# B&R Automation Studio project GAT (part 6)

#### RecipeMgt.typ - Local data types
```iecst
TYPE
	RecipeCommands_type : 	STRUCT
		StoreMachineSettings : BOOL;
		FactoryResetMachineSettings : BOOL;
		SaveCurrentRecipe : BOOL;
		ImportFromUSB : BOOL;
		ExportToUSB : BOOL;
		SaveSelectedRecipe : BOOL;
		LoadRecipe : BOOL;
		CreateRecipe : BOOL;
	END_STRUCT;
	RecipeParameters_type : 	STRUCT
		Category : STRING[30];
		LastLoadedConfigRecipe : STRING[255];
		LastLoadedProductRecipe : STRING[255];
		ActiveRecipe : STRING[255];
		DeviceDataProvider : ARRAY[0..MAX_IDX_FILE_DEV]OF STRING[100];
		DeviceName : STRING[50];
		FileName : STRING[255];
		LastSelectedIndex : UINT;
		LastStatus : MpRecipeUIStatusEnum;
		TableConfig : STRING[120];
		CopyStep : RecipeCopyStep_enum;
		CategoryDropdown : STRING[50];
		EditDialogOpened : BOOL;
		CreateDialogOpened : BOOL;
	END_STRUCT;
	RecipeStatus_type : 	STRUCT
		HMIcommand : RecipeHmiStep_enum;
	END_STRUCT;
	RecipeHmiInterface_type : 	STRUCT
		Commands : RecipeCommands_type;
		Parameters : RecipeParameters_type;
		Status : RecipeStatus_type;
	END_STRUCT;
	RecipeCopyStep_enum :
		(
		REC_COPY_WAIT := 0,
		REC_COPY_TO_USB,
		REC_COPY_FROM_USB,
		REC_COPY_BUSY
		);
	MachineSettings_type : 	STRUCT
		AddMachineSettingsHere1 : USINT;
		AddMachineSettingsHere2 : DINT;
		AddMachineSettingsHere3 : BOOL;
		AddMachineSettingsHere4 : REAL;
		AddMachineSettingsHere5 : UINT;
	END_STRUCT;
	Parameters_type : 	STRUCT
		AddParametersHere1 : BOOL;
		AddParametersHere2 : STRING[80];
		AddParametersHere3 : REAL;
		AddParametersHere4 : REAL;
		AddParametersHere5 : REAL;
	END_STRUCT;
	RecipeHmiStep_enum :
		(
		REC_HMI_WAIT,
		REC_HMI_LOAD,
		REC_HMI_SAVE,
		REC_HMI_CREATE
		);
END_TYPE
```

#### RecipeMgt.var - Local variables
```iecst
(********************************************************************
 * COPYRIGHT -- Bernecker + Rainer
 ********************************************************************
 * Program: FolderHandling
 * File: FolderHandling.var
 * Author: Bernecker + Rainer
 * Created: December , 2020
 ********************************************************************
 * Local variables of program AlarmManagement
 ********************************************************************)
(*Function Block Declaration*)
VAR
	MpRecipe_0 : MpRecipeXml; (*Recipe Management Function Block*)
	MpRecipeUI_0 : MpRecipeUI; (*Recipe to UI*)
	DirCreate_New : DirCreate;
END_VAR
(*Recipe Management Variables*)
VAR
	Index : USINT; (*Index to loop through file devices*)
	MpRecipeUISetup : MpRecipeUISetupType; (*MpRecipeUI connection datapoints*) (*ParameterFileStep : INT;*)
	MpRecipeUIConnect : MpRecipeUIConnectType; (*MpRecipeUI connection datapoints*) (*ParameterFileStep : INT;*)
	HmiRecipe : RecipeHmiInterfaceType;
	Header : MpRecipeXmlHeaderType;
	DTGetTime_0 : DTGetTime;
END_VAR
(*File Management Variables*)
VAR
	MpFileManagerUIConnect : MpFileManagerUIConnectType;
	MpFileManagerUI_0 : MpFileManagerUI;
END_VAR
(*Defines*)
VAR CONSTANT
	MAX_IDX_FILE_DEV : USINT := MAX_IDX_USB_DEV_LIST + 1;
	MACHINE_FILENAME : STRING[12] := 'Machine.mcfg';
	LOCAL_FOLDER : STRING[10] := 'Recipe';
END_VAR
VAR
	MpRecipeRegPar_PreviewPar : MpRecipeRegPar;
	MpRecipeRegPar_PreviewCfg : MpRecipeRegPar;
	Parameters : ParametersType;
	ParametersEdit : {REDUND_UNREPLICABLE} ParametersType;
	ParametersPreview : ParametersType;
	MachineSettings : MachineSettingsType;
	MachineSettingsEdit : MachineSettingsType;
	MachineSettingsPreview : MachineSettingsType;
	PreviousRecipe : STRING[80];
END_VAR
```

#### HMIActions.st
```iecst
ACTION FormatDeviceDataProvider:

	// Select CF device if USB device is not available
	FOR Index := 0 TO MAX_IDX_USB_DEV_LIST DO
		IF gUSBAvailable[Index] THEN
			HmiRecipe.Parameters.DeviceDataProvider[Index + 1] := '{"value":"USB';
			brsitoa(Index + 1, ADR(HmiRecipe.Parameters.DeviceDataProvider[Index + 1]) + brsstrlen(ADR(HmiRecipe.Parameters.DeviceDataProvider[Index + 1])));
			brsstrcat(ADR(HmiRecipe.Parameters.DeviceDataProvider[Index + 1]), ADR('","text":"USB'));
			brsitoa(Index + 1, ADR(HmiRecipe.Parameters.DeviceDataProvider[Index + 1]) + brsstrlen(ADR(HmiRecipe.Parameters.DeviceDataProvider[Index + 1])));
			brsstrcat(ADR(HmiRecipe.Parameters.DeviceDataProvider[Index + 1]), ADR('"}'));
			brsstrcpy(ADR(MpFileManagerUIConnect.DeviceList.DeviceNames[Index + 1]), ADR('USB'));
			brsitoa(Index + 1, ADR(MpFileManagerUIConnect.DeviceList.DeviceNames[Index + 1]) + brsstrlen(ADR(MpFileManagerUIConnect.DeviceList.DeviceNames[Index + 1])));
		ELSE
			brsmemset(ADR(HmiRecipe.Parameters.DeviceDataProvider[Index + 1]), 0, SIZEOF(HmiRecipe.Parameters.DeviceDataProvider[Index + 1]));
			brsmemset(ADR(MpFileManagerUIConnect.DeviceList.DeviceNames[Index + 1]), 0, SIZEOF(MpFileManagerUIConnect.DeviceList.DeviceNames[Index + 1]));
		END_IF
	END_FOR

	// Configure visible recipe list
	HmiRecipe.Parameters.TableConfig := '{ "specRows": [{"from":';
	brsitoa(MpRecipeUIConnect.Recipe.List.MaxSelection + 1, ADR(HmiRecipe.Parameters.TableConfig) + brsstrlen(ADR(HmiRecipe.Parameters.TableConfig)));
	brsstrcat(ADR(HmiRecipe.Parameters.TableConfig),  ADR(',"to":19, "visible":false}]}'));

END_ACTION

ACTION LoadPreview:

	// Load preview when a recipe is selected
	IF (MpRecipeUIConnect.Recipe.List.SelectedIndex <> HmiRecipe.Parameters.LastSelectedIndex) THEN
		// Check selected recipe name is not empty
		IF (brsstrlen(ADR(MpRecipeUIConnect.Recipe.List.Names[MpRecipeUIConnect.Recipe.List.SelectedIndex])) > 0) THEN
			MpRecipe_0.FileName := ADR(MpRecipeUIConnect.Recipe.List.Names[MpRecipeUIConnect.Recipe.List.SelectedIndex]);
			MpRecipe_0.Category := ADR(HmiRecipe.Parameters.CategoryDropdown);
			MpRecipe_0.Load := TRUE;
			HmiRecipe.Parameters.LastSelectedIndex := MpRecipeUIConnect.Recipe.List.SelectedIndex;
		END_IF
	END_IF

	// Reset load command on MpRecipe_Pre FUB
	IF ((MpRecipe_0.CommandDone = TRUE) OR (MpRecipe_0.Error = TRUE)) THEN
		MpRecipe_0.Load := FALSE;
	END_IF

END_ACTION

ACTION RecipeHMIcommands:

    CASE HmiRecipe.Status.HMIcommand OF
        REC_HMI_WAIT:
            IF HmiRecipe.Commands.CreateRecipe THEN
				HmiRecipe.Status.HMIcommand := REC_HMI_CREATE;
				HmiRecipe.Commands.CreateRecipe := FALSE;
			ELSIF HmiRecipe.Commands.SaveSelectedRecipe THEN
				HmiRecipe.Status.HMIcommand := REC_HMI_SAVE;
				HmiRecipe.Commands.SaveSelectedRecipe := FALSE;
			ELSIF HmiRecipe.Commands.LoadRecipe THEN
				HmiRecipe.Status.HMIcommand := REC_HMI_LOAD;
				HmiRecipe.Commands.LoadRecipe := FALSE;
			END_IF

		REC_HMI_CREATE:
			IF (brsstrcmp(ADR(HmiRecipe.Parameters.CategoryDropdown),ADR('Product')) = 0) THEN
				ParametersPreview := ParametersEdit;
			ELSIF (brsstrcmp(ADR(HmiRecipe.Parameters.CategoryDropdown),ADR('Machine')) = 0) THEN
				MachSettingsPreview := MachSettingsEdit;
			END_IF
			MpRecipeUIConnect.New.Create := TRUE;
			HmiRecipe.Status.HMIcommand := REC_HMI_WAIT;

		REC_HMI_LOAD:
			IF (brsstrcmp(ADR(HmiRecipe.Parameters.CategoryDropdown),ADR('Product')) = 0) THEN
				Parameters := ParametersPreview;
				HmiRecipe.Parameters.LastLoadedProductRecipe := HmiRecipe.Parameters.ActiveRecipe;
			ELSIF (brsstrcmp(ADR(HmiRecipe.Parameters.CategoryDropdown),ADR('Machine')) = 0) THEN
				MachSettings := MachSettingsPreview;
				HmiRecipe.Parameters.LastLoadedConfigRecipe := HmiRecipe.Parameters.ActiveRecipe;
			END_IF
			HmiRecipe.Status.HMIcommand := REC_HMI_WAIT;

		REC_HMI_SAVE:
			IF (brsstrcmp(ADR(HmiRecipe.Parameters.CategoryDropdown),ADR('Product')) = 0) THEN
				ParametersPreview := ParametersEdit;
	        ELSIF (brsstrcmp(ADR(HmiRecipe.Parameters.CategoryDropdown),ADR('Machine')) = 0) THEN
                MachSettingsPreview := MachSettingsEdit;
            END_IF

            IF (brsstrlen(ADR(HmiRecipe.Parameters.ActiveRecipe)) > 0) THEN
                MpRecipe_0.FileName := ADR(HmiRecipe.Parameters.ActiveRecipe);
				MpRecipe_0.Save := TRUE;
			END_IF
			HmiRecipe.Status.HMIcommand := REC_HMI_WAIT;

	END_CASE

	IF NOT MpRecipe_0.CommandBusy AND brsstrcmp(ADR(PreviousRecipe),ADR(HmiRecipe.Parameters.FileName)) <> 0 THEN
		HmiRecipe.Parameters.FileName := PreviousRecipe;
	END_IF

	IF HmiRecipe.Parameters.EditDialogOpened OR HmiRecipe.Parameters.CreateDialogOpened THEN
		IF (brsstrcmp(ADR(HmiRecipe.Parameters.CategoryDropdown),ADR('Product')) = 0) THEN
			ParametersEdit := ParametersPreview;
			MpRecipeUIConnect.New.FileName := 'newParameters.par';
		ELSIF (brsstrcmp(ADR(HmiRecipe.Parameters.CategoryDropdown),ADR('Machine')) = 0) THEN
			MachSettingsEdit := MachSettingsPreview;
			MpRecipeUIConnect.New.FileName := 'newMachConfig.mcfg';
		END_IF
		HmiRecipe.Parameters.EditDialogOpened := FALSE;
		HmiRecipe.Parameters.CreateDialogOpened := FALSE;
	END_IF

END_ACTION
```

#### FileOperations.st
```iecst
ACTION FileCopyOperation:

	// Export/Import recipes to/from USB
    CASE HmiRecipe.Parameters.CopyStep OF
		REC_COPY_WAIT:
			//Wait for export/import command
            IF (HmiRecipe.Commands.ExportToUSB = TRUE) THEN
                // Check if USB device is available
                IF (brsstrlen(ADR(MpFileManagerUIConnect.DeviceList.DeviceNames[1])) > 0) THEN
					// USB is available proceed with export: select all files on the CF and trigger copy command
                    IF (MpFileManagerUIConnect.DeviceList.SelectedIndex <> 0) THEN
                        MpFileManagerUIConnect.DeviceList.SelectedIndex := 0;
                        MpFileManagerUIConnect.File.MultiSelect := FALSE;
                    ELSIF (MpFileManagerUIConnect.Status = mpFILE_UI_STATUS_IDLE) THEN

                        IF NOT MpFileManagerUIConnect.File.MultiSelect THEN
                            MpFileManagerUIConnect.File.MultiSelect := TRUE;
                            FOR Index := 0 TO 49 DO
                                MpFileManagerUIConnect.File.List.Items[Index].IsSelected := TRUE;
                            END_FOR
                        ELSIF (brsstrlen(ADR(MpFileManagerUIConnect.File.List.Items[Index].Name)) = 0) THEN
                            // No files to copy, cancel operation
                            HmiRecipe.Commands.ExportToUSB := FALSE;
                        ELSE
                            MpFileManagerUIConnect.File.Copy := TRUE;
							HmiRecipe.Parameters.CopyStep := REC_COPY_TO_USB;
                            HmiRecipe.Commands.ExportToUSB := FALSE;
                        END_IF

                    END_IF

                ELSE
                    // No USB disk available, cancel operation
                    HmiRecipe.Commands.ExportToUSB := FALSE;
                END_IF

            ELSIF HmiRecipe.Commands.ImportFromUSB THEN
                // Check if USB device is available
                IF (brsstrlen(ADR(MpFileManagerUIConnect.DeviceList.DeviceNames[1])) > 0) THEN
                    // USB is available proceed with import: select all files on the USB and trigger copy command

                    IF (MpFileManagerUIConnect.DeviceList.SelectedIndex <> 1) THEN
                        MpFileManagerUIConnect.DeviceList.SelectedIndex := 1;
                        MpFileManagerUIConnect.File.MultiSelect := FALSE;
                    ELSIF MpFileManagerUIConnect.Status = mpFILE_UI_STATUS_IDLE THEN

                        IF NOT MpFileManagerUIConnect.File.MultiSelect THEN
                            MpFileManagerUIConnect.File.MultiSelect := TRUE;
                            FOR Index := 0 TO ((SIZEOF(MpFileManagerUIConnect.File.List.Items)/SIZEOF(MpFileManagerUIConnect.File.List.Items[0])) - 1) DO
                                MpFileManagerUIConnect.File.List.Items[Index].IsSelected := TRUE;
                            END_FOR
                        ELSIF (brsstrlen(ADR(MpFileManagerUIConnect.File.List.Items[Index].Name)) = 0) THEN
                            // No files to copy, cancel operation
                            HmiRecipe.Commands.ImportFromUSB := FALSE;
                        ELSE
                            MpFileManagerUIConnect.File.Copy := TRUE;
                            HmiRecipe.Parameters.CopyStep := REC_COPY_FROM_USB;
                            HmiRecipe.Commands.ImportFromUSB := FALSE;
                        END_IF

                    END_IF
                ELSE
                    // No USB disk available, cancel operation
                    HmiRecipe.Commands.ImportFromUSB := FALSE;
                END_IF

            END_IF

		REC_COPY_TO_USB:
			//Navigate to USB device and paste files
            IF (MpFileManagerUIConnect.Status = mpFILE_UI_STATUS_IDLE) THEN

                IF (MpFileManagerUIConnect.DeviceList.SelectedIndex <> 1) THEN
                    MpFileManagerUIConnect.DeviceList.SelectedIndex := 1;
                    MpFileManagerUIConnect.File.MultiSelect := FALSE;
                ELSE
                    MpFileManagerUIConnect.File.Paste := TRUE;
                END_IF

            END_IF

            IF MpFileManagerUIConnect.Status = mpFILE_UI_STATUS_PASTE THEN
                HmiRecipe.Parameters.CopyStep := REC_COPY_BUSY;
            END_IF

		REC_COPY_FROM_USB:
			//Navigate to CF device and paste files
            IF (MpFileManagerUIConnect.DeviceList.SelectedIndex <> 0) THEN
                MpFileManagerUIConnect.DeviceList.SelectedIndex := 0;
                MpFileManagerUIConnect.File.MultiSelect := FALSE;
            ELSIF (MpFileManagerUIConnect.Status = mpFILE_UI_STATUS_IDLE) THEN
                MpFileManagerUIConnect.File.Paste := TRUE;
            END_IF

            IF (MpFileManagerUIConnect.Status = mpFILE_UI_STATUS_PASTE) THEN
                HmiRecipe.Parameters.CopyStep := REC_COPY_BUSY;
            END_IF

		REC_COPY_BUSY:
			//Wait for copying done
            IF (MpFileManagerUIConnect.MessageBox.Type = mpFILE_MSG_CONFIRM_OVERWRITE) OR (MpFileManagerUIConnect.MessageBox.Type = mpFILE_MSG_BUSY) THEN
                // TODO: Replace by confirm dialog
                MpFileManagerUIConnect.MessageBox.Confirm := TRUE;
            ELSIF MpFileManagerUIConnect.Status = mpFILE_UI_STATUS_IDLE THEN
                MpRecipeUIConnect.Recipe.Refresh := (MpRecipeUIConnect.Status = mpRECIPE_UI_STATUS_IDLE);
                HmiRecipe.Parameters.CopyStep := REC_COPY_WAIT;
            END_IF

    END_CASE

END_ACTION
```

#### MachineSettings.st - not listed in the package file held
```iecst
ACTION MachineSettings:

	// Handle recipe commands
    IF ((hmiRecipe.Commands.StoreMachineSettings = TRUE) AND (MpRecipeUIConnect.Status = mpRECIPE_UI_STATUS_IDLE)) THEN
        // Store factory settings
        hmiRecipe.Commands.StoreMachineSettings := FALSE;
        brsstrcpy(ADR(hmiRecipe.Parameters.Category), ADR(MACHINE_CATEGORY));
        brsstrcpy(ADR(hmiRecipe.Parameters.FileName), ADR(MACHINE_FILENAME));
        DTGetTime_0(enable := TRUE);
        Header.DateTime := DTGetTime_0.DT1;
        Header.Name := MACHINE_FILENAME;
        Header.Description := 'Machine Settings';
        MpRecipe_0.Save := TRUE;
    ELSIF ((hmiRecipe.Commands.FactoryResetMachineSettings = TRUE) AND (MpRecipeUIConnect.Status = mpRECIPE_UI_STATUS_IDLE)) THEN
        // Factory reset the machine settings
        brsstrcpy(ADR(hmiRecipe.Parameters.Category), ADR(MACHINE_CATEGORY));
        brsstrcpy(ADR(hmiRecipe.Parameters.FileName), ADR(MACHINE_FILENAME));
        MpRecipe_0.Load := TRUE;

        IF MpRecipe_0.CommandDone THEN
            // Copy factory settings into Machine.fix file
            hmiRecipe.Commands.FactoryResetMachineSettings := FALSE;
            hmiRecipe.Commands.StoreMachineSettings := TRUE;
        END_IF
    END_IF

END_ACTION
```

#### PreviewOperations.st - not listed in the package file held
```iecst
ACTION LoadPreview:

	(* Load preview when a recipe is selected *)
    IF ((MpRecipeUIConnect.Recipe.List.SelectedIndex <> hmiRecipe.Intern.LastSelectedIndex) AND (MpRecipeXml_Pre.Active = TRUE)) THEN
        (* Check selected recipe name is not empty *)

        IF (brsstrlen(ADR(MpRecipeUIConnect.Recipe.List.Names[MpRecipeUIConnect.Recipe.List.SelectedIndex])) > 0) THEN
            MpRecipeXml_Pre.Load := TRUE;
            MpRecipeXml_Pre.FileName := ADR(MpRecipeUIConnect.Recipe.List.Names[MpRecipeUIConnect.Recipe.List.SelectedIndex]);
            hmiRecipe.Intern.LastSelectedIndex := MpRecipeUIConnect.Recipe.List.SelectedIndex;
        END_IF

    END_IF

    (* Reset load command on MpRecipe_Pre FUB *)
    IF ((MpRecipeXml_Pre.CommandDone = TRUE) OR (MpRecipeXml_Pre.Error = TRUE)) THEN
        MpRecipeXml_Pre.Load := FALSE;
    END_IF;

END_ACTION
```

### Package Logical/Infrastructure/UserX - Package for mapp UserX Framework

### Program Logical/Infrastructure/UserX/UserXMgr (IEC) - UserX manager

#### UserXMgr.st - Init, cyclic, exit code
```iecst
//***********************************************************************
// Copyright: B&R Industrial Automation GmbH
// Author: B&R Industrial Automation GmbH
// Created: Jan 1, 2022
// Description: Tasks for user control. The User Management handling is
// done in this task.
//***********************************************************************

PROGRAM _INIT

	// Create folder for this component on the user file device
	DirCreate_0(enable := TRUE, pDevice := ADR('UserPartition'), pName := ADR(LOCAL_FOLDER));

	// Check if folder already exist and if so disabled the function block call
	IF DirCreate_0.status = fiERR_DIR_ALREADY_EXIST THEN
		DirCreate_0(enable := FALSE);
	END_IF

	// Initialize mapp function blocks
	UserXMgrUIConnect.User.Create.Lock := FALSE;
	UserXMgrUIConnect.User.Lock := FALSE;
	UserXMgrUIConnect.User.Edit.Lock := FALSE;
    UserXMgrUIConnect.User.Create.Dialog.UserName := "";
    UserXMgrUIConnect.User.Create.Dialog.NewPassword := "";
	UserXMgrUIConnect.User.Create.Dialog.ConfirmPassword := "";
	UserXMgrUIConnect.User.List.MaxSelection := USER_LIST_MAX_SELECTION;
	UserXMgrUIConnect.User.List.RangeStart := USER_LIST_RANGE_START;
	UserXMgrUIConnect.User.List.RangeEnd := USER_LIST_RANGE_END;
    MpUserXManagerUI_0.MpLink := ADR(gMpLinkUserXLogin);
    MpUserXManagerUI_0.Enable := TRUE;
    MpUserXManagerUI_0.UIConnect := ADR(UserXMgrUIConnect);
	MpUserXManagerUI_0();

	MpUserXLoginUI_0.MpLink := ADR(gMpLinkUserXLogin);
    MpUserXLoginUI_0.Enable := TRUE;
	MpUserXLoginUI_0.UIConnect := ADR(UserXLoginUIConnect);
	MpUserXLoginUI_0();

	MpUserXLogin_0.MpLink := ADR(gMpLinkUserXLogin);
	MpUserXLogin_0.Enable := TRUE;
	MpUserXLogin_0();

END_PROGRAM

PROGRAM _CYCLIC

	// Error reset
	IF NOT MpUserXManagerUI_0.Error THEN
		MpUserXManagerUI_0.ErrorReset := FALSE;
    END_IF

	IF NOT MpUserXLoginUI_0.Error THEN
		MpUserXLoginUI_0.ErrorReset := FALSE;
    END_IF

	IF NOT MpUserXLogin_0.Error THEN
		MpUserXLogin_0.ErrorReset := FALSE;
    END_IF

	// Assign MpLinks
	MpUserXManagerUI_0.MpLink := ADR(gMpLinkUserXLogin);
	MpUserXLoginUI_0.MpLink := ADR(gMpLinkUserXLogin);
	MpUserXLogin_0.MpLink := ADR(gMpLinkUserXLogin);

	// Call function blocks
	MpUserXManagerUI_0();
	MpUserXLoginUI_0();
	MpUserXLogin_0();

END_PROGRAM

PROGRAM _EXIT

	// Disable the function blocls to unlink the MpLinks
    MpUserXManagerUI_0.Enable := FALSE;
	MpUserXLoginUI_0.Enable := FALSE;
	MpUserXLogin_0.Enable := FALSE;

	// Call function blocks
	MpUserXManagerUI_0();
	MpUserXLoginUI_0();
	MpUserXLogin_0();

END_PROGRAM
```

#### UserXMgr.var - Local variables
```iecst
(*Function Blocks*)
VAR
	MpUserXLogin_0 : MpUserXLogin; (*MpUserXLogin instance*)
	MpUserXManagerUI_0 : MpUserXManagerUI := (UISetup:=(FileDevice:='mappUserXFiles')); (*MpUserXManagerUI instance*)
	MpUserXLoginUI_0 : MpUserXLoginUI; (*MpUserXLoginUI instance*)
	DirCreate_0 : DirCreate; (*DirCreate instance*)
END_VAR
(*Constants*)
VAR CONSTANT
	USER_LIST_MAX_SELECTION : USINT := 20; (*Maxiumum selections on the User List *)
	USER_LIST_RANGE_START : USINT := 0; (*Range start (used for UserXMgrUIConnect)*)
	USER_LIST_RANGE_END : USINT := 20; (*Range end (used for UserXMgrUIConnect)*)
	LOCAL_FOLDER : STRING[10] := 'UserX'; (*Folder name on the file device for UserX  files*)
END_VAR
(*Structure Types*)
VAR
	UserXMgrUIConnect : MpUserXMgrUIConnectType; (*UserX manager connection to the HMI*)
	UserXLoginUIConnect : MpUserXLoginUIConnectType; (*UserL login connection to the HMI*)
END_VAR
```

#### GetErrorText.st - not listed in the package file held
```iecst
ACTION GetErrorText:

	IF UserXMgrUIConnect.MessageBox.ErrorNumber <> 0 OR UserXLoginUIConnect.MessageBox.ErrorNumber <> 0 THEN
		IF UserXMgrUIConnect.MessageBox.ErrorNumber =  28672 OR UserXLoginUIConnect.MessageBox.ErrorNumber =  28672 THEN
			ErrorText := '$$IAT/UserMgmt/Error.28672';
		ELSIF UserXMgrUIConnect.MessageBox.ErrorNumber = 28673  OR UserXLoginUIConnect.MessageBox.ErrorNumber =  28673 THEN
			ErrorText := '$$IAT/UserMgmt/Error.28673';
		ELSIF UserXMgrUIConnect.MessageBox.ErrorNumber = 28674 OR UserXLoginUIConnect.MessageBox.ErrorNumber = 28674 THEN
			ErrorText := '$$IAT/UserMgmt/Error.28674';
		ELSIF UserXMgrUIConnect.MessageBox.ErrorNumber = 28676 OR UserXLoginUIConnect.MessageBox.ErrorNumber = 28676 THEN
			ErrorText := '$$IAT/UserMgmt/Error.28676';
		ELSIF UserXMgrUIConnect.MessageBox.ErrorNumber = 28677  OR UserXLoginUIConnect.MessageBox.ErrorNumber = 28677 THEN
			ErrorText := '$$IAT/UserMgmt/Error.28677';
		ELSIF UserXMgrUIConnect.MessageBox.ErrorNumber = 28679 OR UserXLoginUIConnect.MessageBox.ErrorNumber  = 28679 THEN
			ErrorText := '$$IAT/UserMgmt/Error.28679';
		ELSIF UserXMgrUIConnect.MessageBox.ErrorNumber = 28680 OR UserXLoginUIConnect.MessageBox.ErrorNumber = 28680 THEN
			ErrorText := '$$IAT/UserMgmt/Error.28680';
		ELSIF UserXMgrUIConnect.MessageBox.ErrorNumber = 28685 OR UserXLoginUIConnect.MessageBox.ErrorNumber = 28685 THEN
			ErrorText := '$$IAT/UserMgmt/Error.28685';
		ELSIF UserXMgrUIConnect.MessageBox.ErrorNumber = 28698  OR UserXLoginUIConnect.MessageBox.ErrorNumber = 28698 THEN
			ErrorText := '$$IAT/UserMgmt/Error.28698';
		ELSIF UserXMgrUIConnect.MessageBox.ErrorNumber =  28706 OR UserXLoginUIConnect.MessageBox.ErrorNumber = 28706 THEN
			ErrorText := '$$IAT/UserMgmt/Error.28706';
		ELSIF UserXMgrUIConnect.MessageBox.ErrorNumber =  28695  OR UserXLoginUIConnect.MessageBox.ErrorNumber = 28695 THEN
			ErrorText := '$$IAT/UserMgmt/Error.28695';
		ELSIF UserXMgrUIConnect.MessageBox.ErrorNumber =  28672 OR UserXLoginUIConnect.MessageBox.ErrorNumber = 28672 THEN
			ErrorText := '$$IAT/UserMgmt/Error.28672';
		ELSIF UserXMgrUIConnect.MessageBox.ErrorNumber =  0  OR UserXLoginUIConnect.MessageBox.ErrorNumber = 0 THEN
			ErrorText := '$$IAT/UserMgmt/Error.0';
		END_IF
	END_IF

END_ACTION
```

### Program Logical/Infrastructure/UserX/UserXMgt (IEC)

#### UserX.st - Init, cyclic, exit code
```iecst
//***********************************************************************
// Copyright: B&R Industrial Automation GmbH
// Author: B&R Industrial Automation GmbH
// Created: Jan 1, 2022
// Description: Tasks for user control. The User Management handling is
// done in this task.
//***********************************************************************

PROGRAM _INIT
	// Create folder for this component on the user file device
	DirCreate_New(enable := TRUE, pDevice := ADR('userPartition'), pName := ADR(LOCAL_FOLDER));

	// Check if folder already exist and if so disabled the function block call
	IF DirCreate_New.status = fiERR_DIR_ALREADY_EXIST THEN
		DirCreate_New(enable := FALSE);
	END_IF

	// Init MpUserX
	UserXMgrUIConnect.User.Create.Lock := FALSE;
	UserXMgrUIConnect.User.Lock := FALSE;
	UserXMgrUIConnect.User.Edit.Lock := FALSE;
    UserXMgrUIConnect.User.Create.Dialog.UserName := "";
    UserXMgrUIConnect.User.Create.Dialog.NewPassword := "";
    UserXMgrUIConnect.User.Create.Dialog.ConfirmPassword := "";
    MpUserXManagerUI_0.MpLink := ADR(gUserXLoginMpLink);
    MpUserXManagerUI_0.Enable := TRUE;
    MpUserXManagerUI_0.UIConnect := ADR(UserXMgrUIConnect);
    UserXMgrUIConnect.User.List.MaxSelection := USER_LIST_MAX_SELECTION;
    UserXMgrUIConnect.User.List.RangeStart := USER_LIST_RANGE_START;
    UserXMgrUIConnect.User.List.RangeEnd := USER_LIST_RANGE_END;

	MpUserXLoginUI_0.MpLink := ADR(gUserXLoginMpLink);
    MpUserXLoginUI_0.Enable := TRUE;
	MpUserXLoginUI_0.UIConnect := ADR(UserXLoginUIConnect);

	MpUserXLogin_0.MpLink := ADR(gUserXLoginMpLink);
    MpUserXLogin_0.Enable := TRUE;

END_PROGRAM

PROGRAM _CYCLIC

	//Error reset
	IF NOT MpUserXManagerUI_0.Error THEN
		MpUserXManagerUI_0.ErrorReset := FALSE;
    END_IF

	IF NOT MpUserXLoginUI_0.Error THEN
		MpUserXLoginUI_0.ErrorReset := FALSE;
    END_IF

	IF NOT MpUserXLogin_0.Error THEN
		MpUserXLogin_0.ErrorReset := FALSE;
    END_IF

	MpUserXManagerUI_0();
	MpUserXLoginUI_0();
	MpUserXLogin_0();

END_PROGRAM

PROGRAM _EXIT

	// Call disbaled mapp function blocks
    MpUserXManagerUI_0.Enable := FALSE;
	MpUserXManagerUI_0();

	MpUserXLoginUI_0.Enable := FALSE;
	MpUserXLoginUI_0();

	MpUserXLogin_0.Enable := FALSE;
	MpUserXLogin_0();

END_PROGRAM
```

#### UserX.var - Local variables
```iecst
(********************************************************************
 * COPYRIGHT -- Bernecker + Rainer
 ********************************************************************
 * Program: FolderHandling
 * File: FolderHandling.var
 * Author: Bernecker + Rainer
 * Created: December , 2020
 ********************************************************************
 * Local variables of program User Management
 ********************************************************************)
(*UserX Function Blocks-----------------------------------------------------------------------------------------------------------*)
VAR
	MpUserXManagerUI_0 : MpUserXManagerUI := (UISetup:=(FileDevice:='mappUserX')); (*Management of User X in UI*)
	UserXMgrUIConnect : MpUserXMgrUIConnectType; (*Setup of UserX to UI*)
	MpUserXLoginUI_0 : MpUserXLoginUI;
	UserXLoginUIConnect : MpUserXLoginUIConnectType;
	DirCreate_New : DirCreate;
	MpUserXLogin_0 : MpUserXLogin;
END_VAR
(*UserX Related Variables--------------------------------------------------------------------------------------------------------*)
(*Constants---------------------------------------------------------------------------------------------------------------------------------*)
VAR CONSTANT
	USER_LIST_MAX_SELECTION : USINT := 20; (*Maxiumum Selections on the User List*)
	USER_LIST_RANGE_START : USINT := 0;
	USER_LIST_RANGE_END : USINT := 20;
	LOCAL_FOLDER : STRING[10] := 'UserX';
END_VAR
```

#### UserXFunctions.st
```iecst
// --------------------------------------------------------------------------------------------------------------------
// Create mappView data provider string
FUNCTION String2DataProvider
	brsstrcpy(TargetString, ADR('{"value":"'));
	brsstrcat(TargetString, SourceString);
	brsstrcat(TargetString, ADR('","text":"'));
	brsstrcat(TargetString, SourceString);
	brsstrcat(TargetString, ADR('"}'));
	String2DataProvider := TRUE;
END_FUNCTION
```

#### UserXMgt.var - not listed in the package file held
```iecst
(********************************************************************
 * COPYRIGHT -- Bernecker + Rainer
 ********************************************************************
 * Program: FolderHandling
 * File: FolderHandling.var
 * Author: Bernecker + Rainer
 * Created: December , 2020
 ********************************************************************
 * Local variables of program User Management
 ********************************************************************)
(*UserX Function Blocks*)
VAR
	MpUserXManagerUI_0 : MpUserXManagerUI := (UISetup:=(FileDevice:='mappUserXFiles')); (*Management of User X in UI*)
	UserXMgrUIConnect : MpUserXMgrUIConnectType; (*Setup of UserX to UI*)
	MpUserXLoginUI_0 : MpUserXLoginUI;
	UserXLoginUIConnect : MpUserXLoginUIConnectType;
	DirCreate_New : DirCreate;
	MpUserXLogin_0 : MpUserXLogin;
END_VAR
(*UserX Related Variables*)
(*Constants*)
VAR CONSTANT
	USER_LIST_MAX_SELECTION : USINT := 20; (*Maxiumum Selections on the User List*)
	USER_LIST_RANGE_START : USINT := 0;
	USER_LIST_RANGE_END : USINT := 20;
	LOCAL_FOLDER : STRING[10] := 'UserX';
END_VAR
```

#### UserXMgt.st - not listed in the package file held
```iecst
//***********************************************************************
// Copyright: B&R Industrial Automation GmbH
// Author: B&R Industrial Automation GmbH
// Created: Jan 1, 2022
// Description: Tasks for user control. The User Management handling is
// done in this task.
//***********************************************************************

PROGRAM _INIT

	// Create folder for this component on the user file device
	DirCreate_New(enable := TRUE, pDevice := ADR('userPartition'), pName := ADR(LOCAL_FOLDER));

	// Check if folder already exist and if so disabled the function block call
	IF DirCreate_New.status = fiERR_DIR_ALREADY_EXIST THEN
		DirCreate_New(enable := FALSE);
	END_IF

	// Initialize mapp function blocks
	UserXMgrUIConnect.User.Create.Lock := FALSE;
	UserXMgrUIConnect.User.Lock := FALSE;
	UserXMgrUIConnect.User.Edit.Lock := FALSE;
    UserXMgrUIConnect.User.Create.Dialog.UserName := "";
    UserXMgrUIConnect.User.Create.Dialog.NewPassword := "";
	UserXMgrUIConnect.User.Create.Dialog.ConfirmPassword := "";
	UserXMgrUIConnect.User.List.MaxSelection := USER_LIST_MAX_SELECTION;
	UserXMgrUIConnect.User.List.RangeStart := USER_LIST_RANGE_START;
	UserXMgrUIConnect.User.List.RangeEnd := USER_LIST_RANGE_END;
    MpUserXManagerUI_0.MpLink := ADR(gMpLinkUserXLogin);
    MpUserXManagerUI_0.Enable := TRUE;
    MpUserXManagerUI_0.UIConnect := ADR(UserXMgrUIConnect);
	MpUserXManagerUI_0();

	MpUserXLoginUI_0.MpLink := ADR(gMpLinkUserXLogin);
    MpUserXLoginUI_0.Enable := TRUE;
	MpUserXLoginUI_0.UIConnect := ADR(UserXLoginUIConnect);
	MpUserXLoginUI_0();

	MpUserXLogin_0.MpLink := ADR(gMpLinkUserXLogin);
	MpUserXLogin_0.Enable := TRUE;
	MpUserXLogin_0();

END_PROGRAM

PROGRAM _CYCLIC

	// Error reset
	IF NOT MpUserXManagerUI_0.Error THEN
		MpUserXManagerUI_0.ErrorReset := FALSE;
    END_IF

	IF NOT MpUserXLoginUI_0.Error THEN
		MpUserXLoginUI_0.ErrorReset := FALSE;
    END_IF

	IF NOT MpUserXLogin_0.Error THEN
		MpUserXLogin_0.ErrorReset := FALSE;
    END_IF

	// Assign MpLinks
	MpUserXManagerUI_0.MpLink := ADR(gMpLinkUserXLogin);
	MpUserXLoginUI_0.MpLink := ADR(gMpLinkUserXLogin);
	MpUserXLogin_0.MpLink := ADR(gMpLinkUserXLogin);

	// Call function blocks
	MpUserXManagerUI_0();
	MpUserXLoginUI_0();
	MpUserXLogin_0();

END_PROGRAM

PROGRAM _EXIT

	// Disable the function blocls to unlink the MpLinks
    MpUserXManagerUI_0.Enable := FALSE;
	MpUserXLoginUI_0.Enable := FALSE;
	MpUserXLogin_0.Enable := FALSE;

	// Call function blocks
	MpUserXManagerUI_0();
	MpUserXLoginUI_0();
	MpUserXLogin_0();

END_PROGRAM
```

### Package Logical/Infrastructure/Backup - Package for mapp Backup Framework

### Program Logical/Infrastructure/Backup/BackupMgr (IEC)

#### BackupMgr.st - Init, cyclic, exit code
```iecst
//***********************************************************************
// Copyright: B&R Industrial Automation GmbH
// Author: B&R Industrial Automation GmbH
// Created: April 12, 2022
// Description: Task for backup management.
//***********************************************************************

PROGRAM _INIT

	// Create folder for this component on the user file device
	DirCreate_0(enable := TRUE, pDevice := ADR('UserPartition'), pName := ADR(LOCAL_FOLDER));

	// Check if folder already exist and if so disabled the function block call
	IF DirCreate_0.status = fiERR_DIR_ALREADY_EXIST THEN
		DirCreate_0(enable := FALSE);
	END_IF

	// Initialize mapp function blocks
    MpBackupCore_0.MpLink := ADR(gMpLinkBackupCore);
	MpBackupCore_0.Enable := TRUE;
	MpBackupCore_0();

    MpFileManagerUI_0.MpLink := ADR(gMpLinkFileManagerUIBackup);
    MpFileManagerUI_0.UIConnect := ADR(MpFileManagerUIConnect);
	MpFileManagerUI_0.Enable := TRUE;
	MpFileManagerUI_0();

    MpBackupCoreConfig_0.Enable := TRUE;
    MpBackupCoreConfig_0.MpLink := ADR(gMpLinkBackupCore);
    MpBackupCoreConfig_0.Configuration := ADR(MpBackupConfiguration);
	MpBackupCoreConfig_0.Load := TRUE;
	MpBackupCoreConfig_0();

	HmiBackup.Status.DeviceDataProvider[0] := '{"value":"mappBackupFiles","text":"CF/PLC"}';

END_PROGRAM

PROGRAM _CYCLIC

    CASE BackupState OF
        BACKUP_IDLE:
            HmiBackup.Status.CreateAllowed := NOT(MpBackupCore_0.Info.Automatic.Backup.InProgress);
            HmiBackup.Status.Busy := FALSE;
            IF (HmiBackup.Commands.Create = TRUE) THEN
                HmiBackup.Commands.Create := FALSE;
                MpBackupCore_0.Create := TRUE;
                HmiBackup.Status.Busy := TRUE;
                HmiBackup.Status.CreateAllowed := FALSE;
                HmiBackup.Status.RestoreAllowed := FALSE;
                MpBackupCore_0.Name := ADR(HmiBackup.Parameters.Name);
                BackupState := BACKUP_CREATING;
            ELSIF (HmiBackup.Commands.Restore = TRUE) THEN
                HmiBackup.Commands.Restore := FALSE;
                MpBackupCore_0.Install := TRUE;
                HmiBackup.Status.Busy := TRUE;
                HmiBackup.Status.CreateAllowed := FALSE;
                HmiBackup.Status.RestoreAllowed := FALSE;
                MpBackupCore_0.Name := ADR(MpFileManagerUIConnect.File.List.Items[HmiBackup.Status.SelectedIndex].Name);
                BackupState := BACKUP_RESTORING;
			ELSIF (HmiBackup.Commands.Delete = TRUE) THEN
				MpFileManagerUIConnect.File.List.Items[HmiBackup.Status.SelectedIndex].IsSelected := TRUE;
				HmiBackup.Commands.Delete := FALSE;
				MpFileManagerUIConnect.File.Delete := TRUE;
				BackupState := BACKUP_DELETING;
			ELSIF (HmiBackup.Commands.SaveConfig = TRUE) THEN
				HmiBackup.Commands.SaveConfig := FALSE;
                SaveBackupConfiguration;
                MpBackupCoreConfig_0.Save := TRUE;
			ELSIF ((HmiBackup.Status.SelectedIndex <> HmiBackup.Status.LastSelectedIndex) AND (MpBackupCore_0.CommandBusy <> TRUE)) THEN
                HmiBackup.Status.LastSelectedIndex := HmiBackup.Status.SelectedIndex;
                MpBackupCore_0.Name := ADR(MpFileManagerUIConnect.File.List.Items[HmiBackup.Status.SelectedIndex].Name);
                MpBackupCore_0.RequestInfo := TRUE;
			ELSIF DiagCpuIsARsim() OR DiagCpuIsSimulated() THEN
              	HmiBackup.Status.SimulationActive := TRUE;
                HmiBackup.Status.CreateAllowed := FALSE;
                HmiBackup.Status.RestoreAllowed := FALSE;
            END_IF

        BACKUP_CREATING:
            IF (MpBackupCore_0.CommandDone = TRUE) THEN
				HmiBackup.Status.LastSelectedIndex := HmiBackup.Status.LastSelectedIndex + 1;
                MpBackupCore_0.Create := FALSE;
                MpBackupCore_0.Install := FALSE;
                MpBackupCore_0.RequestInfo := FALSE;
                MpFileManagerUIConnect.File.Refresh := TRUE;
                BackupState := BACKUP_IDLE;
            ELSIF (MpBackupCore_0.Error = TRUE) THEN
                BackupState := BACKUP_ERROR;
                MpBackupCore_0.Create := FALSE;
                MpBackupCore_0.Install := FALSE;
                MpBackupCore_0.RequestInfo := FALSE;
            END_IF

        BACKUP_RESTORING:
            IF (MpBackupCore_0.CommandDone = TRUE) THEN
                MpBackupCore_0.Create := FALSE;
                MpBackupCore_0.Install := FALSE;
                MpBackupCore_0.RequestInfo := FALSE;
                MpFileManagerUIConnect.File.Refresh := TRUE;
                BackupState := BACKUP_IDLE;
            ELSIF (MpBackupCore_0.Error = TRUE) THEN
                BackupState := BACKUP_ERROR;
                MpBackupCore_0.Create := FALSE;
                MpBackupCore_0.Install := FALSE;
                MpBackupCore_0.RequestInfo := FALSE;
            END_IF

        BACKUP_DELETING:
            CASE (MpFileManagerUIConnect.MessageBox.Type) OF
                mpFILE_MSG_CONFIRM_DELETE:
                    MpFileManagerUIConnect.MessageBox.Confirm := TRUE;
                mpFILE_MSG_OK:
                    IF (MpFileManagerUIConnect.Status = mpFILE_UI_STATUS_IDLE) THEN
						HmiBackup.Status.LastSelectedIndex := HmiBackup.Status.LastSelectedIndex + 1;
                        FOR i := 0 TO ((SIZEOF(MpFileManagerUIConnect.File.List.Items[i])/SIZEOF(MpFileManagerUIConnect.File.List.Items[0])) - 1) DO
                            MpFileManagerUIConnect.File.List.Items[i].IsSelected := FALSE;
                        END_FOR
						MpFileManagerUIConnect.MessageBox.Confirm := FALSE;
                        BackupState := BACKUP_IDLE;
                    END_IF
			END_CASE

        BACKUP_ERROR:
			IF MpBackupCore_0.Info.Diag.StatusID.ID = mpBACKUP_ERR_CREATE_FAILED THEN
				HmiBackup.Status.Error := TRUE;
			END_IF
			IF HmiBackup.Commands.Reset THEN
				HmiBackup.Commands.Reset := FALSE;
				MpBackupCore_0.ErrorReset := TRUE;
        		BackupState := BACKUP_IDLE;
			END_IF
    END_CASE

    // Reset any errors caused by requesting information
    IF ((MpBackupCore_0.Error = TRUE) AND (MpBackupCore_0.RequestInfo = TRUE)) THEN
        MpBackupCore_0.ErrorReset := TRUE;
        MpBackupCore_0.RequestInfo := FALSE;
        brsmemset(ADR(HmiBackup.Status.Info), 0, SIZEOF(HmiBackup.Status.Info));
    END_IF
    MpBackupCore_0.MpLink := ADR(gMpLinkBackupCore);
    MpBackupCore_0.DeviceName := ADR(MpFileManagerUIConnect.DeviceList.DeviceNames[MpFileManagerUIConnect.DeviceList.SelectedIndex]);
    MpBackupCore_0();
    IF (MpBackupCore_0.CommandDone = TRUE) AND (MpBackupCore_0.RequestInfo = TRUE) THEN
        MpBackupCore_0.RequestInfo := FALSE;
        HmiBackup.Status.Info := MpBackupCore_0.Info.Project.Requested;
    END_IF
    IF (MpBackupCore_0.Error = FALSE) THEN
        MpBackupCore_0.ErrorReset := FALSE;
		HmiBackup.Status.Error := FALSE;
    END_IF

	HmiBackup.Status.RestoreAllowed := (MpFileManagerUIConnect.File.PathInfo.FolderCount > 0) AND NOT(MpBackupCore_0.Info.Automatic.Backup.InProgress);

	// Call all actions
    FileManager;
	ChangeConfiguration;
	FormatDeviceDataProvider;

	// Assign MpLinks
	MpBackupCore_0.MpLink := ADR(gMpLinkBackupCore);
	MpFileManagerUI_0.MpLink := ADR(gMpLinkFileManagerUIBackup);
	MpBackupCoreConfig_0.MpLink := ADR(gMpLinkBackupCore);

	// Call function blocks
	MpBackupCore_0();
	MpFileManagerUI_0();
	MpBackupCoreConfig_0();

END_PROGRAM

PROGRAM _EXIT

	// Disable the function blocks to unlink the MpLinks
    MpBackupCore_0.Enable := FALSE;
	MpFileManagerUI_0.Enable := FALSE;
	MpBackupCoreConfig_0.Enable := FALSE;

	// Call function blocks
	MpBackupCore_0();
	MpFileManagerUI_0();
	MpBackupCoreConfig_0();

END_PROGRAM
```

#### BackupMgr.typ - Local data types
```iecst
(*Structure types*)

TYPE
	BackupHmiInterfaceType : 	STRUCT  (*HMI interface structure*)
		Commands : BackupHmiCommandsType; (*Structure to hold the commands from the HMI*)
		Parameters : BackupHmiParametersType; (*Structure to hold the parameters for the HMI*)
		Status : BackupHmiStatusType; (*Structure to hold the status information from the HMI*)
	END_STRUCT;
	BackupHmiCommandsType : 	STRUCT  (*Structure to hold the commands from the HMI*)
		Create : BOOL; (*Create a backup*)
		Restore : BOOL; (*Restore a backup*)
		Delete : BOOL; (*Delete a backup*)
		SaveConfig : BOOL; (*Save automatic backup configuration settings*)
		Reset : BOOL; (*Error reset*)
	END_STRUCT;
	BackupHmiParametersType : 	STRUCT  (*Structure to hold the parameters for the HMI*)
		Name : STRING[80] := 'myBackup'; (*Name of the backup*)
		AutomaticBackup : AutomaticBackupType; (*Automatic backup settings*)
	END_STRUCT;
	BackupHmiStatusType : 	STRUCT  (*Structure to hold the status information from the HMI*)
		Busy : BOOL; (*Backup is busy executing an action*)
		Error : BOOL; (*Error flag*)
		CreateAllowed : BOOL; (*Bit to indicate it is allowable to create a backup right now*)
		RestoreAllowed : BOOL; (*Bit to indicate it is allowable to restore a backup right now*)
		FileNames : ARRAY[0..49]OF STRING[80]; (*Existing backup file names*)
		TimeStamps : ARRAY[0..49]OF DATE_AND_TIME; (*Time stamps for existing backups*)
		Size : REFERENCE TO ARRAY[0..49]OF UDINT; (*Sizes of existing backup files*)
		Info : MpBackupProjectInfoRequestType; (*Project information (name, configuration ID, configuration version)*)
		DeviceDataProvider : ARRAY[0..MAX_IDX_FILE_DEV]OF STRING[100]; (*Data provider for file device dropdown on automatic backup configuration pop-up*)
		TableConfig : ARRAY[0..1]OF STRING[120]; (*Table configuration for the list of available backups*)
		SimulationActive : BOOL; (*Flag for if simulation is active*)
		SelectedIndex : USINT; (*Index of the selected backup file*)
		LastSelectedIndex : USINT; (*Index of the last selected backup file*)
		LastSelectedDeviceIndex : UINT; (*Index of the last selected file device. Compared with MpFileManagerUIConnect.DeviceList.SelectedIndex*)
	END_STRUCT;
	AutomaticBackupType : 	STRUCT  (*Automatic backup settings*)
		Enable : BOOL; (*Enable automatic backup feature*)
		Prefix : STRING[50]; (*Name prefix for each automatic backup file*)
		Device : STRING[255]; (*File device to store the automatic backup*)
		Mode : AutomaticBackupModeType; (*Automatic backup time interval*)
		OverwriteOldest : MpBackupOverwriteOldestType; (*Defines whether older backups should be deleted or not*)
	END_STRUCT;
	AutomaticBackupModeType : 	STRUCT  (*Automatic backup time interval*)
		Interval : AutomaticBackupIntervalEnum; (*Day interval (daily, or a specfiic day of the week)*)
		Hour : USINT; (*Time (hour)*)
		Minute : USINT; (*Time (minutes)*)
	END_STRUCT;
END_TYPE

(*Enumerations*)

TYPE
	AutomaticBackupIntervalEnum :
		( (*Selection for how often to automatically create a backup*)
		BACKUP_EVERYDAY, (*Every day*)
		BACKUP_MONDAY, (*Every Monday*)
		BACKUP_TUESDAY, (*Every Tuesday*)
		BACKUP_WEDNESDAY, (*Every Wednesday*)
		BACKUP_THURSDAY, (*Every Thursday*)
		BACKUP_FRIDAY, (*Every Friday*)
		BACKUP_SATURDAY, (*Every Saturday*)
		BACKUP_SUNDAY (*Every Sunday*)
		);
	BackupStateEnum :
		( (*States for backup state machine*)
		BACKUP_IDLE, (*Wait state*)
		BACKUP_CREATING, (*Creating a backup*)
		BACKUP_RESTORING, (*Restoring a backup*)
		BACKUP_DELETING, (*Deleting a backup*)
		BACKUP_ERROR (*Error state*)
		);
END_TYPE
```

#### BackupMgr.var - Local variables
```iecst
(*Function Blocks*)
VAR
	MpBackupCore_0 : MpBackupCore; (*MpBackupCore instance*)
	MpBackupCoreConfig_0 : MpBackupCoreConfig; (*MpBackupCoreConfig instance*)
	MpFileManagerUI_0 : MpFileManagerUI; (*MpFileManagerUI instance*)
	DirCreate_0 : DirCreate; (*DirCreate instance*)
END_VAR
(*Constants*)
VAR CONSTANT
	LOCAL_FOLDER : STRING[10] := 'Backup'; (*Folder name on the file device for Backup files*)
	MAX_IDX_FILE_DEV : USINT := MAX_IDX_USB_DEV_LIST + 1; (*Maximum number of  file devices *)
END_VAR
(*Structure Types*)
VAR
	MpBackupConfiguration : MpBackupCoreConfigType; (*MpBackup configuration*)
	MpFileManagerUIConnect : MpFileManagerUIConnectType := (DeviceList:=(DeviceNames:=['mappBackupFiles','USB1',8('')])); (*MpFile connection to the HMI*)
	HmiBackup : BackupHmiInterfaceType; (*HMI interface structure*)
END_VAR
(*Enumerations*)
VAR
	BackupState : BackupStateEnum; (*States for backup state machine*)
END_VAR
(*Variables*)
VAR
	i : USINT; (*Index for loops*)
	DeviceCount : USINT; (*Counter for available file devices*)
END_VAR
```

#### HMIActions.st
```iecst
ACTION FormatDeviceDataProvider:

	// Select CF device if USB device is not available
    FOR i := 0 TO MAX_IDX_USB_DEV_LIST DO
        IF gUSBAvailable[i] THEN
			HmiBackup.Status.DeviceDataProvider[i + 1] := '{"value":"USB';
            brsitoa(i + 1, ADR(HmiBackup.Status.DeviceDataProvider[i + 1]) + brsstrlen(ADR(HmiBackup.Status.DeviceDataProvider[i + 1])));
            brsstrcat(ADR(HmiBackup.Status.DeviceDataProvider[i + 1]), ADR('","text":"USB'));
            brsitoa(i + 1, ADR(HmiBackup.Status.DeviceDataProvider[i + 1]) + brsstrlen(ADR(HmiBackup.Status.DeviceDataProvider[i + 1])));
            brsstrcat(ADR(HmiBackup.Status.DeviceDataProvider[i + 1]), ADR('"}'));
			MpFileManagerUIConnect.DeviceList.DeviceNames[i + 1] := 'USB';
            brsitoa(i + 1, ADR(MpFileManagerUIConnect.DeviceList.DeviceNames[i + 1]) + brsstrlen(ADR(MpFileManagerUIConnect.DeviceList.DeviceNames[i + 1])));
        ELSE
            brsmemset(ADR(HmiBackup.Status.DeviceDataProvider[i + 1]), 0, SIZEOF(HmiBackup.Status.DeviceDataProvider[i + 1]));
            brsmemset(ADR(MpFileManagerUIConnect.DeviceList.DeviceNames[i + 1]), 0, SIZEOF(MpFileManagerUIConnect.DeviceList.DeviceNames[i + 1]));
        END_IF
    END_FOR

	// Configure visible device list
	HmiBackup.Status.TableConfig[0] := '{ "specRows": [{"from":';
	FOR i := 0 TO 9 DO
		IF MpFileManagerUIConnect.DeviceList.DeviceNames[i] <> '' THEN
			DeviceCount := i + 1;
		END_IF
	END_FOR
	brsitoa((DeviceCount), ADR(HmiBackup.Status.TableConfig[0]) + brsstrlen(ADR(HmiBackup.Status.TableConfig[0])));
    brsstrcat(ADR(HmiBackup.Status.TableConfig[0]),  ADR(',"to":9, "visible":false}]}'));

	// Configure visible file list
	HmiBackup.Status.TableConfig[1] := '{ "specRows": [{"from":';
    brsitoa((MpFileManagerUIConnect.File.PathInfo.FileCount + MpFileManagerUIConnect.File.PathInfo.FolderCount), ADR(HmiBackup.Status.TableConfig[1]) + brsstrlen(ADR(HmiBackup.Status.TableConfig[1])));
    brsstrcat(ADR(HmiBackup.Status.TableConfig[1]),  ADR(',"to":49, "visible":false}]}'));

END_ACTION

ACTION SaveBackupConfiguration:

    MpBackupConfiguration.AutomaticBackup.Enabled := HmiBackup.Parameters.AutomaticBackup.Enable;
    MpBackupConfiguration.AutomaticBackup.NamePrefix := HmiBackup.Parameters.AutomaticBackup.Prefix;
    MpBackupConfiguration.AutomaticBackup.DeviceName := HmiBackup.Parameters.AutomaticBackup.Device;
    MpBackupConfiguration.AutomaticBackup.OverwriteOldest := HmiBackup.Parameters.AutomaticBackup.OverwriteOldest;
    MpBackupConfiguration.AutomaticBackup.Mode.Time := UDINT_TO_TOD((((USINT_TO_UDINT(HmiBackup.Parameters.AutomaticBackup.Mode.Hour) * 60) + HmiBackup.Parameters.AutomaticBackup.Mode.Minute) * 60) * 1000);
    CASE HmiBackup.Parameters.AutomaticBackup.Mode.Interval OF
        BACKUP_EVERYDAY:
            MpBackupConfiguration.AutomaticBackup.Mode.Interval := mpBACKUP_INTERVAL_DAILY;
        BACKUP_MONDAY:
            MpBackupConfiguration.AutomaticBackup.Mode.Interval := mpBACKUP_INTERVAL_WEEKLY;
            MpBackupConfiguration.AutomaticBackup.Mode.Day := mpBACKUP_DAY_MONDAY;
        BACKUP_TUESDAY:
            MpBackupConfiguration.AutomaticBackup.Mode.Interval := mpBACKUP_INTERVAL_WEEKLY;
            MpBackupConfiguration.AutomaticBackup.Mode.Day := mpBACKUP_DAY_TUESDAY;
        BACKUP_WEDNESDAY:
            MpBackupConfiguration.AutomaticBackup.Mode.Interval := mpBACKUP_INTERVAL_WEEKLY;
            MpBackupConfiguration.AutomaticBackup.Mode.Day := mpBACKUP_DAY_WEDNESDAY;
        BACKUP_THURSDAY:
            MpBackupConfiguration.AutomaticBackup.Mode.Interval := mpBACKUP_INTERVAL_WEEKLY;
            MpBackupConfiguration.AutomaticBackup.Mode.Day := mpBACKUP_DAY_THURSDAY;
        BACKUP_FRIDAY:
            MpBackupConfiguration.AutomaticBackup.Mode.Interval := mpBACKUP_INTERVAL_WEEKLY;
            MpBackupConfiguration.AutomaticBackup.Mode.Day := mpBACKUP_DAY_FRIDAY;
        BACKUP_SATURDAY:
            MpBackupConfiguration.AutomaticBackup.Mode.Interval := mpBACKUP_INTERVAL_WEEKLY;
            MpBackupConfiguration.AutomaticBackup.Mode.Day := mpBACKUP_DAY_SATURDAY;
        BACKUP_SUNDAY:
            MpBackupConfiguration.AutomaticBackup.Mode.Interval := mpBACKUP_INTERVAL_WEEKLY;
            MpBackupConfiguration.AutomaticBackup.Mode.Day := mpBACKUP_DAY_SUNDAY;
    END_CASE

 END_ACTION

ACTION LoadBackupConfiguration:

    HmiBackup.Parameters.AutomaticBackup.Enable := MpBackupConfiguration.AutomaticBackup.Enabled;
    HmiBackup.Parameters.AutomaticBackup.Prefix := MpBackupConfiguration.AutomaticBackup.NamePrefix;
    HmiBackup.Parameters.AutomaticBackup.Device := MpBackupConfiguration.AutomaticBackup.DeviceName;
    HmiBackup.Parameters.AutomaticBackup.OverwriteOldest := MpBackupConfiguration.AutomaticBackup.OverwriteOldest;
    HmiBackup.Parameters.AutomaticBackup.Mode.Hour := UDINT_TO_USINT(TOD_TO_UDINT(MpBackupConfiguration.AutomaticBackup.Mode.Time) / 1000 / 60 / 60);
    HmiBackup.Parameters.AutomaticBackup.Mode.Minute := UDINT_TO_USINT(TOD_TO_UDINT(MpBackupConfiguration.AutomaticBackup.Mode.Time) / 1000 / 60) - (HmiBackup.Parameters.AutomaticBackup.Mode.Hour * 60);
    CASE MpBackupConfiguration.AutomaticBackup.Mode.Interval OF
        mpBACKUP_INTERVAL_DAILY:
            HmiBackup.Parameters.AutomaticBackup.Mode.Interval := BACKUP_EVERYDAY;
        mpBACKUP_INTERVAL_WEEKLY:
            CASE MpBackupConfiguration.AutomaticBackup.Mode.Day OF
                mpBACKUP_DAY_MONDAY:
                    HmiBackup.Parameters.AutomaticBackup.Mode.Interval := BACKUP_MONDAY;
                mpBACKUP_DAY_TUESDAY:
                    HmiBackup.Parameters.AutomaticBackup.Mode.Interval := BACKUP_TUESDAY;
                mpBACKUP_DAY_WEDNESDAY:
                    HmiBackup.Parameters.AutomaticBackup.Mode.Interval := BACKUP_WEDNESDAY;
                mpBACKUP_DAY_THURSDAY:
                    HmiBackup.Parameters.AutomaticBackup.Mode.Interval := BACKUP_THURSDAY;
                mpBACKUP_DAY_FRIDAY:
                    HmiBackup.Parameters.AutomaticBackup.Mode.Interval := BACKUP_FRIDAY;
                mpBACKUP_DAY_SATURDAY:
                    HmiBackup.Parameters.AutomaticBackup.Mode.Interval := BACKUP_SATURDAY;
                mpBACKUP_DAY_SUNDAY:
                    HmiBackup.Parameters.AutomaticBackup.Mode.Interval := BACKUP_SUNDAY;
            END_CASE
    END_CASE
END_ACTION

ACTION FileManager:

    MpFileManagerUI_0.MpLink := ADR(gMpLinkFileManagerUIBackup);
    MpFileManagerUI_0.UIConnect := ADR(MpFileManagerUIConnect);
    MpFileManagerUI_0();
    FOR i := 0 TO ((SIZEOF(HmiBackup.Status.FileNames)/SIZEOF(HmiBackup.Status.FileNames[0])) - 1) DO
        HmiBackup.Status.FileNames[i] := MpFileManagerUIConnect.File.List.Items[i].Name;
        HmiBackup.Status.TimeStamps[i] := MpFileManagerUIConnect.File.List.Items[i].LastModified;
        HmiBackup.Status.Size[i] := MpFileManagerUIConnect.File.List.Items[i].Size;
    END_FOR

    IF ((MpFileManagerUIConnect.DeviceList.SelectedIndex <> HmiBackup.Status.LastSelectedDeviceIndex) AND (MpFileManagerUIConnect.Status = mpFILE_UI_STATUS_IDLE)) THEN
        HmiBackup.Status.LastSelectedDeviceIndex := MpFileManagerUIConnect.DeviceList.SelectedIndex;
        HmiBackup.Status.LastSelectedIndex := HmiBackup.Status.LastSelectedIndex + 1;
    END_IF

END_ACTION
```

#### ChangeConfiguration.st
```iecst
ACTION ChangeConfiguration:

    MpBackupCoreConfigFB.MpLink := ADR(gMpLinkBackupCore);
    MpBackupCoreConfigFB.Configuration := ADR(MpBackupConfiguration);
    IF (MpBackupCoreConfigFB.Error = TRUE) THEN
        // Loading currently always throws an error about failed to write Auditing.Type
        IF (MpBackupCoreConfigFB.StatusID = mpBACKUP_ERR_CONFIG_LOAD) THEN
            LoadBackupConfiguration;
        END_IF

        MpBackupCoreConfigFB.Load := FALSE;
        MpBackupCoreConfigFB.Save := FALSE;
        MpBackupCoreConfigFB.ErrorReset := TRUE;
    END_IF
    MpBackupCoreConfigFB();
    MpBackupCoreConfigFB.ErrorReset := FALSE;
    IF (MpBackupCoreConfigFB.CommandDone = TRUE) THEN
        IF (MpBackupCoreConfigFB.Load = TRUE) THEN
            LoadBackupConfiguration;
        END_IF
        MpBackupCoreConfigFB.Load := FALSE;
        MpBackupCoreConfigFB.Save := FALSE;
    END_IF

END_ACTION
```

#### BackupMgt.typ - not listed in the package file held
```iecst
TYPE
	AutomaticBackupIntervalEnum :
		(
		BACKUP_EVERYDAY,
		BACKUP_MONDAY,
		BACKUP_TUESDAY,
		BACKUP_WEDNESDAY,
		BACKUP_THURSDAY,
		BACKUP_FRIDAY,
		BACKUP_SATURDAY,
		BACKUP_SUNDAY
		);
	AutomaticBackupModeType : 	STRUCT
		Interval : AutomaticBackupIntervalEnum;
		Hour : USINT;
		Minute : USINT;
	END_STRUCT;
	AutomaticBackupType : 	STRUCT
		Enable : BOOL;
		Prefix : STRING[50];
		Device : STRING[255];
		Mode : AutomaticBackupModeType;
		OverwriteOldest : MpBackupOverwriteOldestType;
	END_STRUCT;
	BackupHmiCommandsType : 	STRUCT
		Create : BOOL;
		RestoreAuto : BOOL;
		Restore : BOOL;
		Delete : BOOL;
		CopyToUSB : BOOL;
		CopyFromUSB : BOOL;
		SaveConfig : BOOL;
	END_STRUCT;
	BackupHmiParametersType : 	STRUCT
		Name : STRING[80] := 'myBackup';
		SelectedIndex : USINT;
		AutomaticBackup : AutomaticBackupType;
	END_STRUCT;
	BackupHmiStatusType : 	STRUCT
		Busy : BOOL;
		CreateAllowed : BOOL;
		RestoreAllowed : BOOL;
		FileNames : ARRAY[0..49]OF STRING[80];
		TimeStamps : ARRAY[0..49]OF DATE_AND_TIME;
		Size : ARRAY[0..49]OF UDINT;
		Info : MpBackupProjectInfoRequestType;
		DeviceDataProvider : ARRAY[0..MAX_IDX_FILE_DEV]OF STRING[100];
		TableConfig : ARRAY[0..1]OF STRING[120];
	END_STRUCT;
	BackupHmiInterfaceType : 	STRUCT
		Commands : BackupHmiCommandsType;
		Parameters : BackupHmiParametersType;
		Status : BackupHmiStatusType;
	END_STRUCT;
	BackupStateEnum :
		(
		BACKUP_IDLE,
		BACKUP_CREATING,
		BACKUP_RESTORING,
		BACKUP_DELETING,
		BACKUP_ERROR
		);
END_TYPE
```

#### BackupMgt.st - not listed in the package file held
```iecst
//***********************************************************************
// Copyright: B&R Industrial Automation GmbH
// Author: B&R Industrial Automation GmbH
// Created: Jan 1, 2022
// Description: Tasks for backup control.
//***********************************************************************

PROGRAM _INIT

	// Create folder for this component on the user file device
	DirCreate_New(enable := TRUE, pDevice := ADR('userPartition'), pName := ADR(LOCAL_FOLDER));

	// Check if folder already exist and if so disabled the function block call
	IF DirCreate_New.status = fiERR_DIR_ALREADY_EXIST THEN
		DirCreate_New(enable := FALSE);
	END_IF

    MpBackupCoreFB.MpLink := ADR(gMpLinkBackupCore);
	MpBackupCoreFB.Enable := TRUE;
	MpBackupCoreFB();

    MpFileManagerUIFB.MpLink := ADR(gMpLinkFileManagerUIBackup);
    MpFileManagerUIFB.UIConnect := ADR(MpFileManagerUIConnect);
	MpFileManagerUIFB.Enable := TRUE;
	MpFileManagerUIFB();

    MpBackupCoreConfigFB.Enable := TRUE;
    MpBackupCoreConfigFB.MpLink := ADR(gMpLinkBackupCore);
    MpBackupCoreConfigFB.Configuration := ADR(HmiBackup.Parameters.AutomaticBackup);
	MpBackupCoreConfigFB.Load := TRUE;
	MpBackupCoreConfigFB();

	HmiBackup.Status.DeviceDataProvider[0] := '{"value":"mappBackupFiles","text":"CF/PLC"}';

END_PROGRAM

PROGRAM _CYCLIC

    CASE BackupState OF
        BACKUP_IDLE:
            HmiBackup.Status.CreateAllowed := NOT(MpBackupCoreFB.Info.Automatic.Backup.InProgress);
            HmiBackup.Status.Busy := FALSE;
            IF (HmiBackup.Commands.Create = TRUE) THEN
                HmiBackup.Commands.Create := FALSE;
                MpBackupCoreFB.Create := TRUE;
                HmiBackup.Status.Busy := TRUE;
                HmiBackup.Status.CreateAllowed := FALSE;
                HmiBackup.Status.RestoreAllowed := FALSE;
                MpBackupCoreFB.Name := ADR(HmiBackup.Parameters.Name);
                BackupState := BACKUP_CREATING;
            ELSIF (HmiBackup.Commands.Restore = TRUE) THEN
                HmiBackup.Commands.Restore := FALSE;
                MpBackupCoreFB.Install := TRUE;
                HmiBackup.Status.Busy := TRUE;
                HmiBackup.Status.CreateAllowed := FALSE;
                HmiBackup.Status.RestoreAllowed := FALSE;
                MpBackupCoreFB.Name := ADR(MpFileManagerUIConnect.File.List.Items[HmiBackup.Parameters.SelectedIndex].Name);
                BackupState := BACKUP_RESTORING;
            ELSIF (HmiBackup.Commands.RestoreAuto = TRUE) THEN
                HmiBackup.Commands.RestoreAuto := FALSE;
                MpBackupCoreFB.Install := TRUE;
                HmiBackup.Status.Busy := TRUE;
                HmiBackup.Status.CreateAllowed := FALSE;
                HmiBackup.Status.RestoreAllowed := FALSE;
                MpBackupCoreFB.Name := ADR(MpBackupCoreFB.Info.Automatic.Update.Name);
                BackupState := BACKUP_RESTORING;
            ELSIF (HmiBackup.Commands.Delete = TRUE) THEN
                MpFileManagerUIConnect.File.List.Items[HmiBackup.Parameters.SelectedIndex].IsSelected := TRUE;
                HmiBackup.Commands.Delete := FALSE;
                MpFileManagerUIConnect.File.Delete := TRUE;
                BackupState := BACKUP_DELETING;
            ELSIF (HmiBackup.Commands.SaveConfig = TRUE) THEN
                HmiBackup.Commands.SaveConfig := FALSE;
                SaveBackupConfiguration;
                MpBackupCoreConfigFB.Save := TRUE;
            ELSIF ((HmiBackup.Parameters.SelectedIndex <> LastSelectedIndex) AND (MpBackupCoreFB.CommandBusy <> TRUE)) THEN
                LastSelectedIndex := HmiBackup.Parameters.SelectedIndex;
                MpBackupCoreFB.Name := ADR(MpFileManagerUIConnect.File.List.Items[HmiBackup.Parameters.SelectedIndex].Name);
                MpBackupCoreFB.RequestInfo := TRUE;
            END_IF

        BACKUP_CREATING:
            IF (MpBackupCoreFB.CommandDone = TRUE) THEN
				LastSelectedIndex := LastSelectedIndex + 1;
                MpBackupCoreFB.Create := FALSE;
                MpBackupCoreFB.Install := FALSE;
                MpBackupCoreFB.RequestInfo := FALSE;
                MpFileManagerUIConnect.File.Refresh := TRUE;
                BackupState := BACKUP_IDLE;
            ELSIF (MpBackupCoreFB.Error = TRUE) THEN
                BackupState := BACKUP_ERROR;
                MpBackupCoreFB.Create := FALSE;
                MpBackupCoreFB.Install := FALSE;
                MpBackupCoreFB.RequestInfo := FALSE;
            END_IF

        BACKUP_RESTORING:
            IF (MpBackupCoreFB.CommandDone = TRUE) THEN
                MpBackupCoreFB.Create := FALSE;
                MpBackupCoreFB.Install := FALSE;
                MpBackupCoreFB.RequestInfo := FALSE;
                MpFileManagerUIConnect.File.Refresh := TRUE;
                BackupState := BACKUP_IDLE;
            ELSIF (MpBackupCoreFB.Error = TRUE) THEN
                BackupState := BACKUP_ERROR;
                MpBackupCoreFB.Create := FALSE;
                MpBackupCoreFB.Install := FALSE;
                MpBackupCoreFB.RequestInfo := FALSE;
            END_IF

        BACKUP_DELETING:
            CASE (MpFileManagerUIConnect.MessageBox.Type) OF
                mpFILE_MSG_CONFIRM_DELETE:
                    MpFileManagerUIConnect.MessageBox.Confirm := TRUE;
                mpFILE_MSG_OK:
                    IF (MpFileManagerUIConnect.Status = mpFILE_UI_STATUS_IDLE) THEN
						LastSelectedIndex := LastSelectedIndex + 1;
                        FOR i := 0 TO ((SIZEOF(MpFileManagerUIConnect.File.List.Items[i])/SIZEOF(MpFileManagerUIConnect.File.List.Items[0])) - 1) DO
                            MpFileManagerUIConnect.File.List.Items[i].IsSelected := FALSE;
                        END_FOR
						MpFileManagerUIConnect.MessageBox.Confirm := FALSE;
                        BackupState := BACKUP_IDLE;
                    END_IF
			END_CASE

        BACKUP_ERROR:

    END_CASE

    // Reset any errors caused by requesting information
    IF ((MpBackupCoreFB.Error = TRUE) AND (MpBackupCoreFB.RequestInfo = TRUE)) THEN
        MpBackupCoreFB.ErrorReset := TRUE;
        MpBackupCoreFB.RequestInfo := FALSE;
        brsmemset(ADR(HmiBackup.Status.Info), 0, SIZEOF(HmiBackup.Status.Info));
    END_IF
    MpBackupCoreFB.MpLink := ADR(gMpLinkBackupCore);
    MpBackupCoreFB.DeviceName := ADR(MpFileManagerUIConnect.DeviceList.DeviceNames[MpFileManagerUIConnect.DeviceList.SelectedIndex]);
    MpBackupCoreFB();
    IF (MpBackupCoreFB.CommandDone = TRUE) AND (MpBackupCoreFB.RequestInfo = TRUE) THEN
        MpBackupCoreFB.RequestInfo := FALSE;
        HmiBackup.Status.Info := MpBackupCoreFB.Info.Project.Requested;
    END_IF
    IF (MpBackupCoreFB.Error = FALSE) THEN
        MpBackupCoreFB.ErrorReset := FALSE;
    END_IF

    HmiBackup.Status.RestoreAllowed := (HmiBackup.Status.Info.ConfigurationID <> '') AND NOT(MpBackupCoreFB.Info.Automatic.Backup.InProgress);

	// Call all actions
    FileManager;
	ChangeConfiguration;
	FormatDeviceDataProvider;

	// Assign MpLinks
	MpBackupCoreFB.MpLink := ADR(gMpLinkBackupCore);
	MpFileManagerUIFB.MpLink := ADR(gMpLinkFileManagerUIBackup);
	MpBackupCoreConfigFB.MpLink := ADR(gMpLinkBackupCore);

	// Call function blocks
	MpBackupCoreFB();
	MpFileManagerUIFB();
	MpBackupCoreConfigFB();

END_PROGRAM

PROGRAM _EXIT

	// Disable the function blocls to unlink the MpLinks
    MpBackupCoreFB.Enable := FALSE;
	MpFileManagerUIFB.Enable := FALSE;
	MpBackupCoreConfigFB.Enable := FALSE;

	// Call function blocks
	MpBackupCoreFB();
	MpFileManagerUIFB();
	MpBackupCoreConfigFB();

END_PROGRAM
```

### Program Logical/Infrastructure/Backup/BackupMgt (IEC)

#### BackupMgt.st - Init, cyclic, exit code
```iecst
//***********************************************************************
// Copyright: B&R Industrial Automation GmbH
// Author: B&R Industrial Automation GmbH
// Created: Jan 1, 2022
// Description: Tasks for backup control.
//***********************************************************************

PROGRAM _INIT

	// Create folder for this component on the user file device
	DirCreate_New(enable := TRUE, pDevice := ADR('userPartition'), pName := ADR(LOCAL_FOLDER));

	// Check if folder already exist and if so disabled the function block call
	IF DirCreate_New.status = fiERR_DIR_ALREADY_EXIST THEN
		DirCreate_New(enable := FALSE);
	END_IF

    MpBackupCoreFB.MpLink := ADR(gMpLinkBackupCore);
	MpBackupCoreFB.Enable := TRUE;
	MpBackupCoreFB();

    MpFileManagerUIFB.MpLink := ADR(gMpLinkFileManagerUIBackup);
    MpFileManagerUIFB.UIConnect := ADR(MpFileManagerUIConnect);
	MpFileManagerUIFB.Enable := TRUE;
	MpFileManagerUIFB();

    MpBackupCoreConfigFB.Enable := TRUE;
    MpBackupCoreConfigFB.MpLink := ADR(gMpLinkBackupCore);
    MpBackupCoreConfigFB.Configuration := ADR(HmiBackup.Parameters.AutomaticBackup);
	MpBackupCoreConfigFB.Load := TRUE;
	MpBackupCoreConfigFB();

	HmiBackup.Status.DeviceDataProvider[0] := '{"value":"mappBackup","text":"CF/PLC"}';

END_PROGRAM

PROGRAM _CYCLIC

    CASE BackupState OF
        BACKUP_IDLE:
            HmiBackup.Status.CreateAllowed := NOT(MpBackupCoreFB.Info.Automatic.Backup.InProgress);
            HmiBackup.Status.Busy := FALSE;
            IF (HmiBackup.Commands.Create = TRUE) THEN
                HmiBackup.Commands.Create := FALSE;
                MpBackupCoreFB.Create := TRUE;
                HmiBackup.Status.Busy := TRUE;
                HmiBackup.Status.CreateAllowed := FALSE;
                HmiBackup.Status.RestoreAllowed := FALSE;
                MpBackupCoreFB.Name := ADR(HmiBackup.Parameters.Name);
                BackupState := BACKUP_CREATING;
            ELSIF (HmiBackup.Commands.Restore = TRUE) THEN
                HmiBackup.Commands.Restore := FALSE;
                MpBackupCoreFB.Install := TRUE;
                HmiBackup.Status.Busy := TRUE;
                HmiBackup.Status.CreateAllowed := FALSE;
                HmiBackup.Status.RestoreAllowed := FALSE;
                MpBackupCoreFB.Name := ADR(MpFileManagerUIConnect.File.List.Items[HmiBackup.Parameters.SelectedIndex].Name);
                BackupState := BACKUP_RESTORING;
            ELSIF (HmiBackup.Commands.RestoreAuto = TRUE) THEN
                HmiBackup.Commands.RestoreAuto := FALSE;
                MpBackupCoreFB.Install := TRUE;
                HmiBackup.Status.Busy := TRUE;
                HmiBackup.Status.CreateAllowed := FALSE;
                HmiBackup.Status.RestoreAllowed := FALSE;
                MpBackupCoreFB.Name := ADR(MpBackupCoreFB.Info.Automatic.Update.Name);
                BackupState := BACKUP_RESTORING;
            ELSIF (HmiBackup.Commands.Delete = TRUE) THEN
                MpFileManagerUIConnect.File.List.Items[HmiBackup.Parameters.SelectedIndex].IsSelected := TRUE;
                HmiBackup.Commands.Delete := FALSE;
                MpFileManagerUIConnect.File.Delete := TRUE;
                BackupState := BACKUP_DELETING;
            ELSIF (HmiBackup.Commands.SaveConfig = TRUE) THEN
                HmiBackup.Commands.SaveConfig := FALSE;
                SaveBackupConfiguration;
                MpBackupCoreConfigFB.Save := TRUE;
            ELSIF ((HmiBackup.Parameters.SelectedIndex <> LastSelectedIndex) AND (MpBackupCoreFB.CommandBusy <> TRUE)) THEN
                LastSelectedIndex := HmiBackup.Parameters.SelectedIndex;
                MpBackupCoreFB.Name := ADR(MpFileManagerUIConnect.File.List.Items[HmiBackup.Parameters.SelectedIndex].Name);
                MpBackupCoreFB.RequestInfo := TRUE;
            END_IF

        BACKUP_CREATING:
            IF (MpBackupCoreFB.CommandDone = TRUE) THEN
				LastSelectedIndex := LastSelectedIndex + 1;
                MpBackupCoreFB.Create := FALSE;
                MpBackupCoreFB.Install := FALSE;
                MpBackupCoreFB.RequestInfo := FALSE;
                MpFileManagerUIConnect.File.Refresh := TRUE;
                BackupState := BACKUP_IDLE;
            ELSIF (MpBackupCoreFB.Error = TRUE) THEN
                BackupState := BACKUP_ERROR;
                MpBackupCoreFB.Create := FALSE;
                MpBackupCoreFB.Install := FALSE;
                MpBackupCoreFB.RequestInfo := FALSE;
            END_IF

        BACKUP_RESTORING:
            IF (MpBackupCoreFB.CommandDone = TRUE) THEN
                MpBackupCoreFB.Create := FALSE;
                MpBackupCoreFB.Install := FALSE;
                MpBackupCoreFB.RequestInfo := FALSE;
                MpFileManagerUIConnect.File.Refresh := TRUE;
                BackupState := BACKUP_IDLE;
            ELSIF (MpBackupCoreFB.Error = TRUE) THEN
                BackupState := BACKUP_ERROR;
                MpBackupCoreFB.Create := FALSE;
                MpBackupCoreFB.Install := FALSE;
                MpBackupCoreFB.RequestInfo := FALSE;
            END_IF

        BACKUP_DELETING:
            CASE (MpFileManagerUIConnect.MessageBox.Type) OF
                mpFILE_MSG_CONFIRM_DELETE:
                    MpFileManagerUIConnect.MessageBox.Confirm := TRUE;
                mpFILE_MSG_OK:
                    IF (MpFileManagerUIConnect.Status = mpFILE_UI_STATUS_IDLE) THEN
						LastSelectedIndex := LastSelectedIndex + 1;
                        FOR i := 0 TO ((SIZEOF(MpFileManagerUIConnect.File.List.Items[i])/SIZEOF(MpFileManagerUIConnect.File.List.Items[0])) - 1) DO
                            MpFileManagerUIConnect.File.List.Items[i].IsSelected := FALSE;
                        END_FOR
						MpFileManagerUIConnect.MessageBox.Confirm := FALSE;
                        BackupState := BACKUP_IDLE;
                    END_IF
			END_CASE

        BACKUP_ERROR:

    END_CASE

    // Reset any errors caused by requesting information
    IF ((MpBackupCoreFB.Error = TRUE) AND (MpBackupCoreFB.RequestInfo = TRUE)) THEN
        MpBackupCoreFB.ErrorReset := TRUE;
        MpBackupCoreFB.RequestInfo := FALSE;
        brsmemset(ADR(HmiBackup.Status.Info), 0, SIZEOF(HmiBackup.Status.Info));
    END_IF
    MpBackupCoreFB.MpLink := ADR(gMpLinkBackupCore);
    MpBackupCoreFB.DeviceName := ADR(MpFileManagerUIConnect.DeviceList.DeviceNames[MpFileManagerUIConnect.DeviceList.SelectedIndex]);
    MpBackupCoreFB();
    IF (MpBackupCoreFB.CommandDone = TRUE) AND (MpBackupCoreFB.RequestInfo = TRUE) THEN
        MpBackupCoreFB.RequestInfo := FALSE;
        HmiBackup.Status.Info := MpBackupCoreFB.Info.Project.Requested;
    END_IF
    IF (MpBackupCoreFB.Error = FALSE) THEN
        MpBackupCoreFB.ErrorReset := FALSE;
    END_IF

    HmiBackup.Status.RestoreAllowed := (HmiBackup.Status.Info.ConfigurationID <> '') AND NOT(MpBackupCoreFB.Info.Automatic.Backup.InProgress);

	// Call all actions
    FileManager;
	ChangeConfiguration;
	FormatDeviceDataProvider;

	// Assign MpLinks
	MpBackupCoreFB.MpLink := ADR(gMpLinkBackupCore);
	MpFileManagerUIFB.MpLink := ADR(gMpLinkFileManagerUIBackup);
	MpBackupCoreConfigFB.MpLink := ADR(gMpLinkBackupCore);

	// Call function blocks
	MpBackupCoreFB();
	MpFileManagerUIFB();
	MpBackupCoreConfigFB();

END_PROGRAM

PROGRAM _EXIT

	// Disable the function blocls to unlink the MpLinks
    MpBackupCoreFB.Enable := FALSE;
	MpFileManagerUIFB.Enable := FALSE;
	MpBackupCoreConfigFB.Enable := FALSE;

	// Call function blocks
	MpBackupCoreFB();
	MpFileManagerUIFB();
	MpBackupCoreConfigFB();

END_PROGRAM
```

#### BackupMgt.typ - Local data types
```iecst
TYPE
	AutomaticBackupInterval_enum :
		(
		BACKUP_EVERYDAY,
		BACKUP_MONDAY,
		BACKUP_TUESDAY,
		BACKUP_WEDNESDAY,
		BACKUP_THURSDAY,
		BACKUP_FRIDAY,
		BACKUP_SATURDAY,
		BACKUP_SUNDAY
		);
	AutomaticBackupMode_type : 	STRUCT
		Interval : AutomaticBackupInterval_enum;
		Hour : USINT;
		Minute : USINT;
	END_STRUCT;
	AutomaticBackup_type : 	STRUCT
		Enable : BOOL;
		Prefix : STRING[50];
		Device : STRING[255];
		Mode : AutomaticBackupMode_type;
		OverwriteOldest : MpBackupOverwriteOldestType;
	END_STRUCT;
	BackupHmiCommands_type : 	STRUCT
		Create : BOOL;
		RestoreAuto : BOOL;
		Restore : BOOL;
		Delete : BOOL;
		CopyToUSB : BOOL;
		CopyFromUSB : BOOL;
		SaveConfig : BOOL;
	END_STRUCT;
	BackupHmiParameters_type : 	STRUCT
		Name : STRING[80] := 'myBackup';
		SelectedIndex : USINT;
		AutomaticBackup : AutomaticBackup_type;
	END_STRUCT;
	BackupHmiStatus_type : 	STRUCT
		Busy : BOOL;
		CreateAllowed : BOOL;
		RestoreAllowed : BOOL;
		FileNames : ARRAY[0..49]OF STRING[80];
		TimeStamps : ARRAY[0..49]OF DATE_AND_TIME;
		Size : ARRAY[0..49]OF UDINT;
		Info : MpBackupProjectInfoRequestType;
		DeviceDataProvider : ARRAY[0..MAX_IDX_FILE_DEV]OF STRING[100];
		TableConfig : ARRAY[0..1]OF STRING[120];
	END_STRUCT;
	BackupHmiInterface_type : 	STRUCT
		Commands : BackupHmiCommands_type;
		Parameters : BackupHmiParameters_type;
		Status : BackupHmiStatus_type;
	END_STRUCT;
	BackupState_enum :
		(
		BACKUP_IDLE,
		BACKUP_CREATING,
		BACKUP_RESTORING,
		BACKUP_DELETING,
		BACKUP_ERROR
		);
END_TYPE
```

#### BackupMgt.var - Local variables
```iecst
VAR
	MpBackupConfiguration : MpBackupCoreConfigType;
	MpBackupCoreConfigFB : MpBackupCoreConfig;
	MpFileManagerUIConnect : MpFileManagerUIConnectType := (DeviceList:=(DeviceNames:=['mappBackup','USB1',8('')]));
	MpFileManagerUIFB : MpFileManagerUI;
	DirCreate_New : DirCreate;
	MpBackupCoreFB : MpBackupCore;
	HmiBackup : BackupHmiInterfaceType;
	i : USINT;
	DeviceCount : USINT;
	BackupState : BackupStateEnum;
	LastSelectedIndex : USINT;
	LastSelectedDeviceIndex : UINT;
END_VAR
VAR CONSTANT
	MAX_IDX_FILE_DEV : USINT := MAX_IDX_USB_DEV_LIST + 1;
	LOCAL_FOLDER : STRING[10] := 'Backup';
END_VAR
```

#### HMIActions.st
```iecst
ACTION FormatDeviceDataProvider:

	// Select CF device if USB device is not available
    FOR i := 0 TO MAX_IDX_USB_DEV_LIST DO
        IF gUSBAvailable[i] THEN
            brsstrcpy(ADR(HmiBackup.Status.DeviceDataProvider[i + 1]), ADR('{"value":"USB'));
            brsitoa(i + 1, ADR(HmiBackup.Status.DeviceDataProvider[i + 1]) + brsstrlen(ADR(HmiBackup.Status.DeviceDataProvider[i + 1])));
            brsstrcat(ADR(HmiBackup.Status.DeviceDataProvider[i + 1]), ADR('","text":"USB'));
            brsitoa(i + 1, ADR(HmiBackup.Status.DeviceDataProvider[i + 1]) + brsstrlen(ADR(HmiBackup.Status.DeviceDataProvider[i + 1])));
            brsstrcat(ADR(HmiBackup.Status.DeviceDataProvider[i + 1]), ADR('"}'));
            brsstrcpy(ADR(MpFileManagerUIConnect.DeviceList.DeviceNames[i + 1]), ADR('USB'));
            brsitoa(i + 1, ADR(MpFileManagerUIConnect.DeviceList.DeviceNames[i + 1]) + brsstrlen(ADR(MpFileManagerUIConnect.DeviceList.DeviceNames[i + 1])));
        ELSE
            brsmemset(ADR(HmiBackup.Status.DeviceDataProvider[i + 1]), 0, SIZEOF(HmiBackup.Status.DeviceDataProvider[i + 1]));
            brsmemset(ADR(MpFileManagerUIConnect.DeviceList.DeviceNames[i + 1]), 0, SIZEOF(MpFileManagerUIConnect.DeviceList.DeviceNames[i + 1]));
        END_IF
    END_FOR

	// Configure visible device list
    brsstrcpy(ADR(HmiBackup.Status.TableConfig[0]), ADR('{ "specRows": [{"from":'));
	FOR i := 0 TO 9 DO
		IF MpFileManagerUIConnect.DeviceList.DeviceNames[i] <> '' THEN
			DeviceCount := i + 1;
		END_IF
	END_FOR
	brsitoa((DeviceCount), ADR(HmiBackup.Status.TableConfig[0]) + brsstrlen(ADR(HmiBackup.Status.TableConfig[0])));
    brsstrcat(ADR(HmiBackup.Status.TableConfig[0]),  ADR(',"to":9, "visible":false}]}'));

	// Configure visible file list
    brsstrcpy(ADR(HmiBackup.Status.TableConfig[1]), ADR('{ "specRows": [{"from":'));
    brsitoa((MpFileManagerUIConnect.File.PathInfo.FileCount + MpFileManagerUIConnect.File.PathInfo.FolderCount), ADR(HmiBackup.Status.TableConfig[1]) + brsstrlen(ADR(HmiBackup.Status.TableConfig[1])));
    brsstrcat(ADR(HmiBackup.Status.TableConfig[1]),  ADR(',"to":49, "visible":false}]}'));

END_ACTION

ACTION SaveBackupConfiguration:

    MpBackupConfiguration.AutomaticBackup.Enabled := HmiBackup.Parameters.AutomaticBackup.Enable;
    MpBackupConfiguration.AutomaticBackup.NamePrefix := HmiBackup.Parameters.AutomaticBackup.Prefix;
    MpBackupConfiguration.AutomaticBackup.DeviceName := HmiBackup.Parameters.AutomaticBackup.Device;
    MpBackupConfiguration.AutomaticBackup.OverwriteOldest := HmiBackup.Parameters.AutomaticBackup.OverwriteOldest;
    MpBackupConfiguration.AutomaticBackup.Mode.Time := UDINT_TO_TOD((((USINT_TO_UDINT(HmiBackup.Parameters.AutomaticBackup.Mode.Hour) * 60) + HmiBackup.Parameters.AutomaticBackup.Mode.Minute) * 60) * 1000);
    CASE HmiBackup.Parameters.AutomaticBackup.Mode.Interval OF
        BACKUP_EVERYDAY:
            MpBackupConfiguration.AutomaticBackup.Mode.Interval := mpBACKUP_INTERVAL_DAILY;
        BACKUP_MONDAY:
            MpBackupConfiguration.AutomaticBackup.Mode.Interval := mpBACKUP_INTERVAL_WEEKLY;
            MpBackupConfiguration.AutomaticBackup.Mode.Day := mpBACKUP_DAY_MONDAY;
        BACKUP_TUESDAY:
            MpBackupConfiguration.AutomaticBackup.Mode.Interval := mpBACKUP_INTERVAL_WEEKLY;
            MpBackupConfiguration.AutomaticBackup.Mode.Day := mpBACKUP_DAY_TUESDAY;
        BACKUP_WEDNESDAY:
            MpBackupConfiguration.AutomaticBackup.Mode.Interval := mpBACKUP_INTERVAL_WEEKLY;
            MpBackupConfiguration.AutomaticBackup.Mode.Day := mpBACKUP_DAY_WEDNESDAY;
        BACKUP_THURSDAY:
            MpBackupConfiguration.AutomaticBackup.Mode.Interval := mpBACKUP_INTERVAL_WEEKLY;
            MpBackupConfiguration.AutomaticBackup.Mode.Day := mpBACKUP_DAY_THURSDAY;
        BACKUP_FRIDAY:
            MpBackupConfiguration.AutomaticBackup.Mode.Interval := mpBACKUP_INTERVAL_WEEKLY;
            MpBackupConfiguration.AutomaticBackup.Mode.Day := mpBACKUP_DAY_FRIDAY;
        BACKUP_SATURDAY:
            MpBackupConfiguration.AutomaticBackup.Mode.Interval := mpBACKUP_INTERVAL_WEEKLY;
            MpBackupConfiguration.AutomaticBackup.Mode.Day := mpBACKUP_DAY_SATURDAY;
        BACKUP_SUNDAY:
            MpBackupConfiguration.AutomaticBackup.Mode.Interval := mpBACKUP_INTERVAL_WEEKLY;
            MpBackupConfiguration.AutomaticBackup.Mode.Day := mpBACKUP_DAY_SUNDAY;
    END_CASE

 END_ACTION

ACTION LoadBackupConfiguration:
    HmiBackup.Parameters.AutomaticBackup.Enable := MpBackupConfiguration.AutomaticBackup.Enabled;
    HmiBackup.Parameters.AutomaticBackup.Prefix := MpBackupConfiguration.AutomaticBackup.NamePrefix;
    HmiBackup.Parameters.AutomaticBackup.Device := MpBackupConfiguration.AutomaticBackup.DeviceName;
    HmiBackup.Parameters.AutomaticBackup.OverwriteOldest := MpBackupConfiguration.AutomaticBackup.OverwriteOldest;
    HmiBackup.Parameters.AutomaticBackup.Mode.Hour := UDINT_TO_USINT(TOD_TO_UDINT(MpBackupConfiguration.AutomaticBackup.Mode.Time) / 1000 / 60 / 60);
    HmiBackup.Parameters.AutomaticBackup.Mode.Minute := UDINT_TO_USINT(TOD_TO_UDINT(MpBackupConfiguration.AutomaticBackup.Mode.Time) / 1000 / 60) - (HmiBackup.Parameters.AutomaticBackup.Mode.Hour * 60);
    CASE MpBackupConfiguration.AutomaticBackup.Mode.Interval OF
        mpBACKUP_INTERVAL_DAILY:
            HmiBackup.Parameters.AutomaticBackup.Mode.Interval := BACKUP_EVERYDAY;
        mpBACKUP_INTERVAL_WEEKLY:
            CASE MpBackupConfiguration.AutomaticBackup.Mode.Day OF
                mpBACKUP_DAY_MONDAY:
                    HmiBackup.Parameters.AutomaticBackup.Mode.Interval := BACKUP_MONDAY;
                mpBACKUP_DAY_TUESDAY:
                    HmiBackup.Parameters.AutomaticBackup.Mode.Interval := BACKUP_TUESDAY;
                mpBACKUP_DAY_WEDNESDAY:
                    HmiBackup.Parameters.AutomaticBackup.Mode.Interval := BACKUP_WEDNESDAY;
                mpBACKUP_DAY_THURSDAY:
                    HmiBackup.Parameters.AutomaticBackup.Mode.Interval := BACKUP_THURSDAY;
                mpBACKUP_DAY_FRIDAY:
                    HmiBackup.Parameters.AutomaticBackup.Mode.Interval := BACKUP_FRIDAY;
                mpBACKUP_DAY_SATURDAY:
                    HmiBackup.Parameters.AutomaticBackup.Mode.Interval := BACKUP_SATURDAY;
                mpBACKUP_DAY_SUNDAY:
                    HmiBackup.Parameters.AutomaticBackup.Mode.Interval := BACKUP_SUNDAY;
            END_CASE
    END_CASE
END_ACTION

ACTION FileManager:
    MpFileManagerUIFB.MpLink := ADR(gMpLinkFileManagerUIBackup);
    MpFileManagerUIFB.UIConnect := ADR(MpFileManagerUIConnect);
    MpFileManagerUIFB();
    FOR i := 0 TO ((SIZEOF(HmiBackup.Status.FileNames)/SIZEOF(HmiBackup.Status.FileNames[0])) - 1) DO
        HmiBackup.Status.FileNames[i] := MpFileManagerUIConnect.File.List.Items[i].Name;
        HmiBackup.Status.TimeStamps[i] := MpFileManagerUIConnect.File.List.Items[i].LastModified;
        HmiBackup.Status.Size[i] := MpFileManagerUIConnect.File.List.Items[i].Size;
    END_FOR

    IF ((MpFileManagerUIConnect.DeviceList.SelectedIndex <> LastSelectedDeviceIndex) AND (MpFileManagerUIConnect.Status = mpFILE_UI_STATUS_IDLE)) THEN
        LastSelectedDeviceIndex := MpFileManagerUIConnect.DeviceList.SelectedIndex;
        LastSelectedIndex := LastSelectedIndex + 1;
    END_IF

END_ACTION
```

#### ChangeConfiguration.st
```iecst
ACTION ChangeConfiguration:

    MpBackupCoreConfigFB.MpLink := ADR(gMpLinkBackupCore);
    MpBackupCoreConfigFB.Configuration := ADR(MpBackupConfiguration);
    IF (MpBackupCoreConfigFB.Error = TRUE) THEN
        // Loading currently always throws an error about failed to write Auditing.Type
        IF (MpBackupCoreConfigFB.StatusID = mpBACKUP_ERR_CONFIG_LOAD) THEN
            LoadBackupConfiguration;
        END_IF

        MpBackupCoreConfigFB.Load := FALSE;
        MpBackupCoreConfigFB.Save := FALSE;
        MpBackupCoreConfigFB.ErrorReset := TRUE;
    END_IF
    MpBackupCoreConfigFB();
    MpBackupCoreConfigFB.ErrorReset := FALSE;
    IF (MpBackupCoreConfigFB.CommandDone = TRUE) THEN
        IF (MpBackupCoreConfigFB.Load = TRUE) THEN
            LoadBackupConfiguration;
        END_IF
        MpBackupCoreConfigFB.Load := FALSE;
        MpBackupCoreConfigFB.Save := FALSE;
    END_IF

END_ACTION
```

#### Variables.var - not listed in the package file held
```iecst
VAR
	MpBackupConfiguration : MpBackupCoreConfigType;
	MpBackupCoreConfigFB : MpBackupCoreConfig;
	MpFileManagerUIConnect : MpFileManagerUIConnectType := (DeviceList:=(DeviceNames:=['mappBackup','USB1',8('')]));
	MpFileManagerUIFB : MpFileManagerUI;
	DirCreate_New : DirCreate;
	MpBackupCoreFB : MpBackupCore;
	hmiBackup : BackupHmiInterface_type;
	i : USINT;
	BackupState : BackupState_enum;
	LastSelectedIndex : USINT;
	LastSelectedDeviceIndex : UINT;
END_VAR
VAR CONSTANT
	MAX_IDX_FILE_DEV : USINT := MAX_IDX_USB_DEV_LIST + 1;
	LOCAL_FOLDER : STRING[10] := 'Backup';
END_VAR
```

#### Configuration.st - not listed in the package file held
```iecst
ACTION Configuration:

    MpBackupCoreConfigFB.MpLink := ADR(gBackupCore);
    MpBackupCoreConfigFB.Configuration := ADR(MpBackupConfiguration);
    IF (MpBackupCoreConfigFB.Error = TRUE) THEN
        // loading currently always throws an error about failed to write Auditing.Type
        IF (MpBackupCoreConfigFB.StatusID = mpBACKUP_ERR_CONFIG_LOAD) THEN
            LoadBackupConfiguration;
        END_IF

        MpBackupCoreConfigFB.Load := FALSE;
        MpBackupCoreConfigFB.Save := FALSE;
        MpBackupCoreConfigFB.ErrorReset := TRUE;
    END_IF
    MpBackupCoreConfigFB();
    MpBackupCoreConfigFB.ErrorReset := FALSE;
    IF (MpBackupCoreConfigFB.CommandDone = TRUE) THEN
        IF (MpBackupCoreConfigFB.Load = TRUE) THEN
            LoadBackupConfiguration;
        END_IF
        MpBackupCoreConfigFB.Load := FALSE;
        MpBackupCoreConfigFB.Save := FALSE;
    END_IF

END_ACTION
```

#### Main.st - not listed in the package file held
```iecst
(*********************************************************************************************************************
* Copyright: B&R Industrial Automation GmbH
* Author:    B&R Industrial Automation GmbH
* Description: Tasks for backup control.
*********************************************************************************************************************)

PROGRAM _INIT

	(*Create folder for this component on the user file device*)
	DirCreate_New(enable := TRUE, pDevice := ADR('userPartition'), pName := ADR(LOCAL_FOLDER));

	(*Check if folder already exist and if so disabled the function block call*)
	IF DirCreate_New.status = fiERR_DIR_ALREADY_EXIST THEN
		DirCreate_New(enable := FALSE);
	END_IF

    MpBackupCoreFB.MpLink := ADR(gBackupCore);
    MpBackupCoreFB.Enable := TRUE;

    MpFileManagerUIFB.MpLink := ADR(gBackupFileManagerUIMpLink);
    MpFileManagerUIFB.UIConnect := ADR(MpFileManagerUIConnect);
    MpFileManagerUIFB.Enable := TRUE;

    MpBackupCoreConfigFB.Enable := TRUE;
    MpBackupCoreConfigFB.MpLink := ADR(gBackupCore);
    MpBackupCoreConfigFB.Configuration := ADR(hmiBackup.Parameters.AutomaticBackup);
    MpBackupCoreConfigFB.Load := TRUE;

    brsstrcpy(ADR(hmiBackup.Status.DeviceDataProvider[0]), ADR('{"value":"mappBackup","text":"CF/PLC"}'));

END_PROGRAM

PROGRAM _CYCLIC

    CASE BackupState OF
        BACKUP_IDLE:
            hmiBackup.Status.CreateAllowed := NOT(MpBackupCoreFB.Info.Automatic.Backup.InProgress);
            hmiBackup.Status.Busy := FALSE;
            IF (hmiBackup.Commands.Create = TRUE) THEN
                hmiBackup.Commands.Create := FALSE;
                MpBackupCoreFB.Create := TRUE;
                hmiBackup.Status.Busy := TRUE;
                hmiBackup.Status.CreateAllowed := FALSE;
                hmiBackup.Status.RestoreAllowed := FALSE;
                MpBackupCoreFB.Name := ADR(hmiBackup.Parameters.Name);
                BackupState := BACKUP_CREATING;
            ELSIF (hmiBackup.Commands.Restore = TRUE) THEN
                hmiBackup.Commands.Restore := FALSE;
                MpBackupCoreFB.Install := TRUE;
                hmiBackup.Status.Busy := TRUE;
                hmiBackup.Status.CreateAllowed := FALSE;
                hmiBackup.Status.RestoreAllowed := FALSE;
                MpBackupCoreFB.Name := ADR(MpFileManagerUIConnect.File.List.Items[hmiBackup.Parameters.SelectedIndex].Name);
                BackupState := BACKUP_RESTORING;
            ELSIF (hmiBackup.Commands.RestoreAuto = TRUE) THEN
                hmiBackup.Commands.RestoreAuto := FALSE;
                MpBackupCoreFB.Install := TRUE;
                hmiBackup.Status.Busy := TRUE;
                hmiBackup.Status.CreateAllowed := FALSE;
                hmiBackup.Status.RestoreAllowed := FALSE;
                MpBackupCoreFB.Name := ADR(MpBackupCoreFB.Info.Automatic.Update.Name);
                BackupState := BACKUP_RESTORING;
            ELSIF (hmiBackup.Commands.Delete = TRUE) THEN
                MpFileManagerUIConnect.File.List.Items[hmiBackup.Parameters.SelectedIndex].IsSelected := TRUE;
                hmiBackup.Commands.Delete := FALSE;
                MpFileManagerUIConnect.File.Delete := TRUE;
                BackupState := BACKUP_DELETING;
            ELSIF (hmiBackup.Commands.SaveConfig = TRUE) THEN
                hmiBackup.Commands.SaveConfig := FALSE;
                SaveBackupConfiguration;
                MpBackupCoreConfigFB.Save := TRUE;
            ELSIF ((hmiBackup.Parameters.SelectedIndex <> LastSelectedIndex) AND (MpBackupCoreFB.CommandBusy <> TRUE)) THEN
                LastSelectedIndex := hmiBackup.Parameters.SelectedIndex;
                MpBackupCoreFB.Name := ADR(MpFileManagerUIConnect.File.List.Items[hmiBackup.Parameters.SelectedIndex].Name);
                MpBackupCoreFB.RequestInfo := TRUE;
            END_IF

        BACKUP_CREATING:
            IF (MpBackupCoreFB.CommandDone = TRUE) THEN
                // force the information refresh
                LastSelectedIndex := LastSelectedIndex + 1;
                MpBackupCoreFB.Create := FALSE;
                MpBackupCoreFB.Install := FALSE;
                MpBackupCoreFB.RequestInfo := FALSE;
                MpFileManagerUIConnect.File.Refresh := TRUE;
                BackupState := BACKUP_IDLE;
            ELSIF (MpBackupCoreFB.Error = TRUE) THEN
                BackupState := BACKUP_ERROR;
                MpBackupCoreFB.Create := FALSE;
                MpBackupCoreFB.Install := FALSE;
                MpBackupCoreFB.RequestInfo := FALSE;
            END_IF

        BACKUP_RESTORING:
            IF (MpBackupCoreFB.CommandDone = TRUE) THEN
                MpBackupCoreFB.Create := FALSE;
                MpBackupCoreFB.Install := FALSE;
                MpBackupCoreFB.RequestInfo := FALSE;
                MpFileManagerUIConnect.File.Refresh := TRUE;
                BackupState := BACKUP_IDLE;
            ELSIF (MpBackupCoreFB.Error = TRUE) THEN
                BackupState := BACKUP_ERROR;
                MpBackupCoreFB.Create := FALSE;
                MpBackupCoreFB.Install := FALSE;
                MpBackupCoreFB.RequestInfo := FALSE;
            END_IF

        BACKUP_DELETING:
            CASE (MpFileManagerUIConnect.MessageBox.Type) OF
                mpFILE_MSG_CONFIRM_DELETE:
                    MpFileManagerUIConnect.MessageBox.Confirm := TRUE;
                mpFILE_MSG_OK:
                    IF (MpFileManagerUIConnect.Status = mpFILE_UI_STATUS_IDLE) THEN
                        // force the information refresh
                        LastSelectedIndex := LastSelectedIndex + 1;
                        FOR i:=0 TO ((SIZEOF(MpFileManagerUIConnect.File.List.Items[i])/SIZEOF(MpFileManagerUIConnect.File.List.Items[0]))-1) DO
                            MpFileManagerUIConnect.File.List.Items[i].IsSelected := FALSE;
                        END_FOR

                        MpFileManagerUIConnect.MessageBox.Confirm := FALSE;
                        BackupState := BACKUP_IDLE;
                    END_IF

            END_CASE

        BACKUP_ERROR:

    END_CASE

    // reset any errors caused by requesting information
    IF ((MpBackupCoreFB.Error = TRUE) AND (MpBackupCoreFB.RequestInfo = TRUE)) THEN
        MpBackupCoreFB.ErrorReset := TRUE;
        MpBackupCoreFB.RequestInfo := FALSE;
        brsmemset(ADR(hmiBackup.Status.Info), 0, SIZEOF(hmiBackup.Status.Info));
    END_IF
    MpBackupCoreFB.MpLink := ADR(gBackupCore);
    MpBackupCoreFB.DeviceName := ADR(MpFileManagerUIConnect.DeviceList.DeviceNames[MpFileManagerUIConnect.DeviceList.SelectedIndex]);
    MpBackupCoreFB();
    IF (MpBackupCoreFB.CommandDone = TRUE) AND (MpBackupCoreFB.RequestInfo = TRUE) THEN
        MpBackupCoreFB.RequestInfo := FALSE;
        hmiBackup.Status.Info := MpBackupCoreFB.Info.Project.Requested;
    END_IF
    IF (MpBackupCoreFB.Error = FALSE) THEN
        MpBackupCoreFB.ErrorReset := FALSE;
    END_IF

    hmiBackup.Status.RestoreAllowed := (hmiBackup.Status.Info.ConfigurationID <> '') AND NOT(MpBackupCoreFB.Info.Automatic.Backup.InProgress);

    FileManager;
	ChangeConfiguration;
	FormatDeviceDataProvider;

END_PROGRAM

PROGRAM _EXIT

    MpBackupCoreFB.Enable := FALSE;
    MpBackupCoreFB();

    MpFileManagerUIFB.Enable := FALSE;
    MpFileManagerUIFB();

    MpBackupCoreConfigFB.Enable := FALSE;
    MpBackupCoreConfigFB();

END_PROGRAM
```

### Package Logical/Infrastructure/SysServices - Package For System Services

### Program Logical/Infrastructure/SysServices/SysServs (IEC) - Services for ETH, and time settings

#### Types.typ
```iecst
TYPE
	CpuIoMap_typ : 	STRUCT
		SerialNumber_CPU : UDINT;
		ModuleID_CPU : UINT;
		HardwareVariant : UINT;
		FirmwareVersion : UINT;
		TemperatureCPU : INT;
		TemperatureENV : INT;
		SystemTime : DINT;
		TerminalOK : BOOL;
		TerminalStatus : USINT;
		TerminalTemperatureCPU : INT;
		TerminalLoadCPU0 : USINT;
		TerminalLoadCPU1 : USINT;
	END_STRUCT;
	LanguageSelect : 	STRUCT
		LanguageSelection : ARRAY[0..1]OF STRING[80] := ['en','de'];
		SelectedIndex : INT := 0;
	END_STRUCT;
	EthConfig_type : 	STRUCT
		Ip : STRING[15];
		Gateway : STRING[15];
		SubnetMask : STRING[15];
		Device : STRING[20];
	END_STRUCT;
	ClientInfo_typ : 	STRUCT
		userId : STRING[40];
		ipAddress : STRING[15];
		activityCount : USINT;
		languageId : STRING[10];
		isValid : BOOL;
		currentPageId : STRING[40];
		measurementSystemId : STRING[10];
	END_STRUCT;
END_TYPE
```

#### Variables.var
```iecst
(********************************************************************
 * COPYRIGHT -- Bernecker + Rainer
 ********************************************************************
 * Program: FolderHandling
 * File: FolderHandling.var
 * Author: Bernecker + Rainer
 * Created: December , 2020
 ********************************************************************
 * Local variables of program Visualization Control
 ********************************************************************)
(*Variable Declaration-------------------------------------------------------------------------*)
VAR
	EthConfig : EthConfigType; (*Ethernet configuration*)
	CpuIoMap : CpuIoMapType; (*Cpu IO Mapping*)
	CfgGetSubnetMask_0 : CfgGetSubnetMask; (*GetSubnetMask*)
	CfgGetIPAddr_0 : CfgGetIPAddr; (*GetIPAddr*)
	CfgGetDefaultGateway_0 : CfgGetDefaultGateway; (*GetDefaultGateway*)
	CfgSetSubnetMask_0 : CfgSetSubnetMask; (*GetSubnetMask*)
	CfgSetIPAddr_0 : CfgSetIPAddr; (*GetIPAddr*)
	CfgSetDefaultGateway_0 : CfgSetDefaultGateway; (*GetDefaultGateway*)
	CurrentMode : STRING[80]; (*Current Mode(Simulation/Runtime)*)
	Simulation : BOOL; (*Simulation Mode Flag(1: Simulation 0: Runtime)*)
	ReadEthConfig : BOOL;
	WriteEthConfig : BOOL;
	DTStructureSetTime_0 : DTStructureGetTime;
	DTStructureGetTime_0 : DTStructureSetTime;
	DateTimeCfg : DTStructure; (*Date Structure*)
	ClientInfo : ARRAY[0..MAX_IDX_CLIENTS] OF ClientInfoType;
END_VAR
VAR CONSTANT
	MAX_IDX_CLIENTS : USINT := 3;
END_VAR
```

#### Main.st
```iecst
//*********************************************************************************
//* Copyright: B&R Industrial Automation GmbH
//* Created:   30. Sep 2020/08:00
//* Description: Tasks FOR Visualization control. The HMI handling is done in this task.
//********************************************************************************

PROGRAM _INIT
	// Insert code here

    brsstrcpy(ADR(EthConfig.Device), ADR('IF2'));

    // Configure Ethernet configuration function blocks
    CfgGetIPAddr_0.pDevice := ADR(EthConfig.Device);
    CfgGetDefaultGateway_0.pDevice := ADR(EthConfig.Device);
    CfgGetSubnetMask_0.pDevice := ADR(EthConfig.Device);
    CfgGetIPAddr_0.pIPAddr := ADR(EthConfig.Ip);
    CfgGetDefaultGateway_0.pGateway := ADR(EthConfig.Gateway);
    CfgGetSubnetMask_0.pSubnetMask := ADR(EthConfig.SubnetMask);
    CfgGetIPAddr_0.Len := 16;
    CfgGetDefaultGateway_0.Len := 16;
    CfgGetSubnetMask_0.Len := 16;
    CfgSetIPAddr_0.pDevice := ADR(EthConfig.Device);
	CfgSetDefaultGateway_0.pDevice := ADR(EthConfig.Device);
	CfgSetSubnetMask_0.pDevice := ADR(EthConfig.Device);
	CfgSetIPAddr_0.pIPAddr := ADR(EthConfig.Ip);
	CfgSetDefaultGateway_0.pGateway := ADR(EthConfig.Gateway);
	CfgSetSubnetMask_0.pSubnetMask := ADR(EthConfig.SubnetMask);
	CfgSetIPAddr_0.Option := 1;
	CfgSetDefaultGateway_0.Option := 1;
	CfgSetSubnetMask_0.Option := 1;

	// Read ETHERNET information after booting
	ReadEthConfig := TRUE;

	// Configure Get/Set time function blocks
	DTStructureGetTime_0.pDTStructure := ADR(DateTimeCfg);
	DTStructureSetTime_0.pDTStructure := ADR(DateTimeCfg);

	// Client info
	ClientInfo[0].activityCount := 0;
END_PROGRAM

PROGRAM _CYCLIC
	// Read ethernet information from target
	IF ReadEthConfig THEN
		CfgGetIPAddr_0.enable := TRUE;
		CfgGetDefaultGateway_0.enable := TRUE;
		CfgGetSubnetMask_0.enable := TRUE;
		ReadEthConfig := FALSE;
	END_IF
	// Write ethernet information to target
	IF WriteEthConfig THEN
		CfgSetIPAddr_0.enable := TRUE;
		CfgSetDefaultGateway_0.enable := TRUE;
		CfgSetSubnetMask_0.enable := TRUE;
		WriteEthConfig := FALSE;
	END_IF

	// Call ethernet configuration related function blocks
	CfgGetIPAddr_0();
	CfgGetDefaultGateway_0();
	CfgGetSubnetMask_0();
	CfgSetIPAddr_0();
	CfgSetDefaultGateway_0();
	CfgSetSubnetMask_0();

	// Reset the enable inputs when done
	IF (CfgGetIPAddr_0.status <> ERR_FUB_BUSY) AND (CfgGetIPAddr_0.status <> ERR_FUB_ENABLE_FALSE) THEN
		CfgGetIPAddr_0.enable := FALSE;
	END_IF
	IF (CfgGetDefaultGateway_0.status <> ERR_FUB_BUSY) AND (CfgGetDefaultGateway_0.status <> ERR_FUB_ENABLE_FALSE) THEN
		CfgGetDefaultGateway_0.enable := FALSE;
	END_IF
	IF (CfgGetSubnetMask_0.status <> ERR_FUB_BUSY) AND (CfgGetSubnetMask_0.status <> ERR_FUB_ENABLE_FALSE) THEN
		CfgGetSubnetMask_0.enable := FALSE;
	END_IF
	IF (CfgSetIPAddr_0.status <> ERR_FUB_BUSY) AND (CfgSetIPAddr_0.status <> ERR_FUB_ENABLE_FALSE) THEN
		CfgSetIPAddr_0.enable := FALSE;
	END_IF
	IF (CfgSetDefaultGateway_0.status <> ERR_FUB_BUSY) AND (CfgSetDefaultGateway_0.status <> ERR_FUB_ENABLE_FALSE) THEN
		CfgSetDefaultGateway_0.enable := FALSE;
	END_IF
	IF (CfgSetSubnetMask_0.status <> ERR_FUB_BUSY) AND (CfgSetSubnetMask_0.status <> ERR_FUB_ENABLE_FALSE) THEN
		CfgSetSubnetMask_0.enable := FALSE;
	END_IF

	// Reset time function block enable commands
	IF (DTStructureGetTime_0.status <> ERR_FUB_BUSY) AND (DTStructureGetTime_0.status <> ERR_FUB_ENABLE_FALSE) THEN
		DTStructureGetTime_0.enable := FALSE;
	END_IF
	IF (DTStructureSetTime_0.status <> ERR_FUB_BUSY) AND (DTStructureSetTime_0.status <> ERR_FUB_ENABLE_FALSE) THEN
		DTStructureSetTime_0.enable := FALSE;
	END_IF

	// Call time configuration function blocks
	DTStructureGetTime_0();
	DTStructureSetTime_0();

	IF CpuIoMap.SerialNumber_CPU = 0 THEN
		CurrentMode := 'Simulation Mode' ;
		Simulation := TRUE ;
	ELSE
		CurrentMode := 'Runtime Mode' ;
		Simulation := FALSE ;
	END_IF

END_PROGRAM

PROGRAM _EXIT
	// Insert code here

END_PROGRAM
```

### Program Logical/Infrastructure/SysServices/ProcessConfig (IEC) - Process the configuration of any axis
